// SIMATIC S7-200 project (STEP 7-Micro/WIN), CPU 226 CN REL 02.01

SYMBOL_TABLE 用户定义1
I_ERR1_QX        I4.2
I_ERR1_SF1       I0.0
I_ERR1_SF2       I0.1
I_ERR1_PF        I0.2
I_ERR1_JR        I0.3
I_TEST1_P        I0.4
I_L_ONOFF1       I0.5
I_ERR2_SF1       I0.7
I_ERR2_SF2       I1.0
I_ERR2_PF        I1.1
I_ERR2_JR        I1.2
I_TEST2_P        I1.3
I_L_ONOFF2       I1.4
I_ERR3_SF1       I1.6
I_ERR3_SF2       I1.7
I_ERR3_PF        I2.0
I_ERR3_JR        I2.1
I_TEST3_P        I2.2
I_L_ONOFF3       I2.3
I_ERR4_SF1       I2.5
I_ERR4_SF2       I2.6
I_ERR4_PF        I2.7
I_ERR4_JR        I3.0
I_TEST4_P        I3.1
I_L_ONOFF4       I3.2
I_MODE_CHANGE    I3.3
I_ONOFF1         I3.4
I_ONOFF2         I3.5
I_ONOFF3         I3.6
I_ONOFF4         I3.7
I_ONOFF          I4.0
I_JT             I4.1
I_ERR_WY         I4.5
I_ERR_GAS        I4.6
I_ERR_FIRE       I4.7
AQ_PF2           AQW0
AQ_PF4           AQW4
Q1_SF1           Q0.0
Q1_SF2           Q0.1
Q1_PF            Q0.2
Q1_JR            Q0.3
Q1_LIGHT         Q0.4
Q1_RUN           Q0.5
Q1_FM            Q0.6
Q1_PQ            Q0.7
Q1_KQ            Q1.0
Q2_SF1           Q1.1
Q2_SF2           Q1.2
Q2_PF            Q1.3
Q2_JR            Q1.4
Q2_LIGHT         Q1.5
Q2_RUN           Q1.6
Q2_FM            Q1.7
Q3_SF1           Q2.0
Q3_SF2           Q2.1
Q3_PF            Q2.2
Q3_JR            Q2.3
Q3_LIGHT         Q2.4
Q3_RUN           Q2.5
Q3_FM            Q2.6
Q4_SF1           Q3.0
Q4_SF2           Q3.1
Q4_PF            Q3.2
Q4_JR            Q3.3
Q4_LIGHT         Q3.4
Q4_RUN           Q3.5
Q4_FM            Q3.6
Q_RUN            Q3.7
F_HOUR_FLAG      M0.0
F_DELAY_WRITE    M0.1
F_DISSTART       M0.2
F_DISSTOP        M0.3
F_AUTO           M0.4
F_FILTER         M0.5
F_SAMPLING       M0.6
F_ERR            M0.7
F_NO_HMI         M1.0
F_S_ONOFF        M1.1
F_START          M1.2
F_STOP           M1.3
F_S_PQ           M1.4
F_S_GD           M1.5
F_S_KQ           M1.6
F_S_TOPPQ        M1.7
F_S_M_CHGE       M2.0
F_EN_M_CHGE      M2.1
F_TO_PQ          M2.2
F_TO_GD          M2.3
F_TO_KQ          M2.4
F_TO_TOPPQ       M2.5
F_GD_RESTART     M2.6
F_S_L_BOT_ONOFF  M2.7
F_RESTART_ALL    M3.0
F_ON_GAS         M3.1
F_RESET_START    M3.2
F_RESET_STOP     M3.3
F_RESET_OP_JR    M3.4
F_RESET_PAUSE    M3.5
F_RESET_RESTART  M3.6
F_RESET_RUN      M3.7
F_RESET_OPEN     M4.0
F_GD1            M4.1
F_GD2            M4.2
F_GD3            M4.3
F_GD4            M4.4
F_GD_END         M4.5
F_MODE_CHGE      M4.6
F_CHANGE         M4.7
F_DELAY_O_24     M5.0
F_Q_CHANGE       M5.1
F_S_ONOFF1       M7.0
F_START1         M7.1
F_STOP1          M7.2
F_S_L_ONOFF1     M7.3
F_ERR1           M7.4
F_RUN1           M7.5
F_OPEN1          M7.6
F_FLASH1         M7.7
F_FLASH1_ON      M8.0
F_PQ1_O_3S       M8.1
F_PQ1_O_6S       M8.2
F_PQ1_C_10S      M8.3
F_PQ1_C_5S       M8.4
F_KQ1_O_30S      M8.5
F_KQ1_O_3S       M8.6
F_KQ1_C_10S      M8.7
F_KQ1_C_5S       M9.0
F_PAUSE1         M9.1
F_RESTART1       M9.2
F1_OP_JR         M9.3
F_S_ONOFF2       M10.0
F_START2         M10.1
F_STOP2          M10.2
F_S_L_ONOFF2     M10.3
F_ERR2           M10.4
F_RUN2           M10.5
F_OPEN2          M10.6
F_FLASH2         M10.7
F_FLASH2_ON      M11.0
F_PQ2_O_3S       M11.1
F_PQ2_O_6S       M11.2
F_PQ2_C_10S      M11.3
F_PQ2_C_5S       M11.4
F_KQ2_O_30S      M11.5
F_KQ2_O_3S       M11.6
F_KQ2_C_10S      M11.7
F_KQ2_C_5S       M12.0
F_PAUSE2         M12.1
F_RESTART2       M12.2
F2_OP_JR         M12.3
F_S_ONOFF3       M13.0
F_START3         M13.1
F_STOP3          M13.2
F_S_L_ONOFF3     M13.3
F_ERR3           M13.4
F_RUN3           M13.5
F_OPEN3          M13.6
F_FLASH3         M13.7
F_FLASH3_ON      M14.0
F_PQ3_O_3S       M14.1
F_PQ3_O_6S       M14.2
F_PQ3_C_10S      M14.3
F_PQ3_C_5S       M14.4
F_KQ3_O_30S      M14.5
F_KQ3_O_3S       M14.6
F_KQ3_C_10S      M14.7
F_KQ3_C_5S       M15.0
F_PAUSE3         M15.1
F_RESTART3       M15.2
F3_OP_JR         M15.3
F_S_ONOFF4       M16.0
F_START4         M16.1
F_STOP4          M16.2
F_S_L_ONOFF4     M16.3
F_ERR4           M16.4
F_RUN4           M16.5
F_OPEN4          M16.6
F_FLASH4         M16.7
F_FLASH4_ON      M17.0
F_PQ4_O_3S       M17.1
F_PQ4_O_6S       M17.2
F_PQ4_C_10S      M17.3
F_PQ4_C_5S       M17.4
F_KQ4_O_30S      M17.5
F_KQ4_O_3S       M17.6
F_KQ4_C_10S      M17.7
F_KQ4_C_5S       M18.0
F_PAUSE4         M18.1
F_RESTART4       M18.2
F4_OP_JR         M18.3
F_S_ONOFF5       M19.0
F_START5         M19.1
F_STOP5          M19.2
F_S_L_ONOFF5     M19.3
F_ERR5           M19.4
F_RUN5           M19.5
F_OPEN5          M19.6
F_FLASH5         M19.7
F_FLASH5_ON      M20.0
F_PQ5_O_3S       M20.1
F_PQ5_O_6S       M20.2
F_PQ5_C_10S      M20.3
F_PQ5_C_5S       M20.4
F_KQ5_O_30S      M20.5
F_KQ5_O_3S       M20.6
F_KQ5_C_10S      M20.7
F_KQ5_C_5S       M21.0
F_PAUSE5         M21.1
F_RESTART5       M21.2
F5_OP_JR         M21.3
SYSTEM_ERROR_FLAG M23.2
Comu_Flag1       M23.3
Comu_Flag2       M23.4
Comu_Start       M23.5
Comu_End         M23.6
Real_Time        VW100
TEMP1_1          VW404
TEMP1_2          VW406
TEMP1_3          VW408
TEMP1_4          VW410
TEMP1_5          VW412
TEMP1_6          VW414
TEMP2_1          VW420
TEMP2_2          VW422
TEMP2_3          VW424
TEMP2_4          VW426
TEMP2_5          VW428
TEMP2_6          VW430
TEMP3_1          VW436
TEMP3_2          VW438
TEMP3_3          VW440
TEMP3_4          VW442
TEMP3_5          VW444
TEMP3_6          VW446
TEMP4_1          VW452
TEMP4_2          VW454
TEMP4_3          VW456
TEMP4_4          VW458
TEMP4_5          VW460
TEMP4_6          VW462
TEMP5_1          VW468
TEMP5_2          VW470
TEMP5_3          VW472
TEMP5_4          VW474
TEMP5_5          VW476
TEMP5_6          VW478
TEMP6_1          VW484
TEMP6_2          VW486
TEMP6_3          VW488
TEMP6_4          VW490
TEMP6_5          VW492
TEMP6_6          VW494
TEMP7_1          VW500
TEMP7_2          VW502
TEMP7_3          VW504
TEMP7_4          VW506
TEMP7_5          VW508
TEMP7_6          VW510
TEMP8_1          VW516
TEMP8_2          VW518
TEMP8_3          VW520
TEMP8_4          VW522
TEMP8_5          VW524
TEMP8_6          VW526
TEMP9_1          VW532
TEMP9_2          VW534
TEMP9_3          VW536
TEMP9_4          VW538
TEMP9_5          VW540
TEMP9_6          VW542
TEMP10_1         VW548
TEMP10_2         VW550
TEMP10_3         VW552
TEMP10_4         VW554
TEMP10_5         VW556
TEMP10_6         VW558
TEMP11_1         VW564
TEMP11_2         VW566
TEMP11_3         VW568
TEMP11_4         VW570
TEMP11_5         VW572
TEMP11_6         VW574
TEMP12_1         VW580
TEMP12_2         VW582
TEMP12_3         VW584
TEMP12_4         VW586
TEMP12_5         VW588
TEMP12_6         VW590
TEMP13_1         VW596
TEMP13_2         VW598
TEMP13_3         VW600
TEMP13_4         VW602
TEMP13_5         VW604
TEMP13_6         VW606
TEMP14_1         VW612
TEMP14_2         VW614
TEMP14_3         VW616
TEMP14_4         VW618
TEMP14_5         VW620
TEMP14_6         VW622
TEMP15_1         VW628
TEMP15_2         VW630
TEMP15_3         VW632
TEMP15_4         VW634
TEMP15_5         VW636
TEMP15_6         VW638
TEMP16_1         VW644
TEMP16_2         VW646
TEMP16_3         VW648
TEMP16_4         VW650
TEMP16_5         VW652
TEMP16_6         VW654
T_ERRL           VW700
T_ERRH           VW702
T_SAMPLING       VW704
ADDR_EEP         VW706
TEMP_PQ_H        VW708
TEMP_PQ_L        VW710
TEMP_PQ_ALARM_T1 VW712
TEMP_PQ_ALARM_T2 VW714
TEMP_KQ_H        VW716
TEMP_KQ_L        VW718
TEMP_KQ_ALARM_T1 VW720
TEMP_KQ_ALARM_T2 VW722
TIME_PQ          VW724
TIME_KQ          VW726
TIME_LQ          VW728
DELAY_START      VW730
TIME_DOOR        VW732
TEMP_H           VW754
TEMP_L           VW756
TEMP_T1_ALARM    VW758
TEMP_T2_ALARM    VW760
DELAY_C_PQ       VW762
DELAY_C_KQ       VW764
T_RUN            VW766
DELAY_O_24       VW768
DELAY_FM         VW770
C_ONOFF          VB800
C_ERR_HMI        VB801
C_SAMPLING       VB802
AD_ADDR          VB803
C_KEY            VB804
C_ERR            VB805
C_ERR_FIRE       VB806
C_ERR_WY         VB807
C_ERR_GAS        VB808
C_JT             VB809
C_PQ             VB810
C_GD             VB811
C_KQ             VB812
C_TOPPQ          VB813
C_M_CHGE         VB814
C_L_BOT_ONOFF    VB815
C_GD1            VB816
C_GD2            VB817
C_GD3            VB818
C_GD4            VB819
C_GD_END         VB820
C_ONOFF1         VB821
C_ERR1_QX        VB822
C_ERR1_SF1       VB823
C_ERR1_SF2       VB824
C_ERR1_PF        VB825
C_ERR1_JR        VB826
C_ERR1_T1        VB827
C_ERR1_T2        VB828
C_OVER1_T1       VB829
C_OVER1_T2       VB830
C_TEST1_P        VB831
C_L_ONOFF1       VB832
EX_MODE          VB833
REAL_MODE        VB834
TEMP_MODE        VB835
C_ONOFF2         VB840
C_L_ONOFF2       VB841
C_ERR2_QX        VB842
C_ERR2_SF1       VB843
C_ERR2_SF2       VB844
C_ERR2_PF        VB845
C_ERR2_JR        VB846
C_ERR2_T1        VB847
C_ERR2_T2        VB848
C_OVER2_T1       VB849
C_OVER2_T2       VB850
C_TEST2_P        VB851
C_ONOFF3         VB860
C_L_ONOFF3       VB861
C_ERR3_QX        VB862
C_ERR3_SF1       VB863
C_ERR3_SF2       VB864
C_ERR3_PF        VB865
C_ERR3_JR        VB866
C_ERR3_T1        VB867
C_ERR3_T2        VB868
C_OVER3_T1       VB869
C_OVER3_T2       VB870
C_TEST3_P        VB871
C_ONOFF4         VB880
C_L_ONOFF4       VB881
C_ERR4_QX        VB882
C_ERR4_SF1       VB883
C_ERR4_SF2       VB884
C_ERR4_PF        VB885
C_ERR4_JR        VB886
C_ERR4_T1        VB887
C_ERR4_T2        VB888
C_OVER4_T1       VB889
C_OVER4_T2       VB890
C_TEST4_P        VB891
C_ONOFF5         VB900
C_L_ONOFF5       VB901
C_ERR5_QX        VB902
C_ERR5_SF1       VB903
C_ERR5_SF2       VB904
C_ERR5_PF        VB905
C_ERR5_JR        VB906
C_ERR5_T1        VB907
C_ERR5_T2        VB908
C_OVER5_T1       VB909
C_OVER5_T2       VB910
C_TEST5_P        VB911
MEASURE_MODE     VB914
C_ERR_W1         VW822
C_ERR_W2         VW842
C_ERR_W3         VW862
C_ERR_W4         VW882
C_ERR_W5         VW902
ERR1_1           VB1000
F_ERR1_QX        V1000.0
F_ERR1_SF1       V1000.1
F_ERR1_SF2       V1000.2
F_ERR1_PF        V1000.3
F_ERR1_JR        V1000.4
F_ERR1_P         V1000.5
ERR1_2           VB1001
F_ERR1_T1        V1001.0
F_ERR1_T2        V1001.1
F_OVER1_T1       V1001.2
F_OVER1_T2       V1001.3
ERR2_1           VB1002
F_ERR2_QX        V1002.0
F_ERR2_SF1       V1002.1
F_ERR2_SF2       V1002.2
F_ERR2_PF        V1002.3
F_ERR2_JR        V1002.4
F_ERR2_P         V1002.5
ERR2_2           VB1003
F_ERR2_T1        V1003.0
F_ERR2_T2        V1003.1
F_OVER2_T1       V1003.2
F_OVER2_T2       V1003.3
ERR3_1           VB1004
F_ERR3_QX        V1004.0
F_ERR3_SF1       V1004.1
F_ERR3_SF2       V1004.2
F_ERR3_PF        V1004.3
F_ERR3_JR        V1004.4
F_ERR3_P         V1004.5
ERR3_2           VB1005
F_ERR3_T1        V1005.0
F_ERR3_T2        V1005.1
F_OVER3_T1       V1005.2
F_OVER3_T2       V1005.3
ERR4_1           VB1006
F_ERR4_QX        V1006.0
F_ERR4_SF1       V1006.1
F_ERR4_SF2       V1006.2
F_ERR4_PF        V1006.3
F_ERR4_JR        V1006.4
F_ERR4_P         V1006.5
ERR4_2           VB1007
F_ERR4_T1        V1007.0
F_ERR4_T2        V1007.1
F_OVER4_T1       V1007.2
F_OVER4_T2       V1007.3
ERR5_1           VB1008
F_ERR5_QX        V1008.0
F_ERR5_SF1       V1008.1
F_ERR5_SF2       V1008.2
F_ERR5_PF        V1008.3
F_ERR5_JR        V1008.4
F_ERR5_P         V1008.5
ERR5_2           VB1009
F_ERR5_T1        V1009.0
F_ERR5_T2        V1009.1
F_OVER5_T1       V1009.2
F_OVER5_T2       V1009.3
EN_QX            VB1010
F_EN_QX1         V1010.0
F_EN_QX2         V1010.1
F_EN_QX3         V1010.2
F_EN_QX4         V1010.3
F_EN_QX5         V1010.4
EN_OP1           VB1011
F_EN_ON_ALL      V1011.0
F_EN_OFF_ALL     V1011.1
F_EN_ON_1        V1011.2
F_EN_OFF_1       V1011.3
F_EN_ON_2        V1011.4
F_EN_OFF_2       V1011.5
F_EN_ON_3        V1011.6
F_EN_OFF_3       V1011.7
EN_OP2           VB1012
F_EN_ON_4        V1012.0
F_EN_OFF_4       V1012.1
F_EN_ON_5        V1012.2
F_EN_OFF_5       V1012.3
STATE            VB1014
F_STATE1         V1014.0
F_STATE2         V1014.1
F_STATE3         V1014.2
F_STATE4         V1014.3
F_STATE5         V1014.4
MINUTE           VB1016
ERR_MOUDLE       VB1017
F_ERR_MK1        V1017.0
F_ERR_MK2        V1017.1
F_ERR_MK3        V1017.2
F_ERR_MK4        V1017.3
F_ERR_MK5        V1017.4
F_ERR_MK6        V1017.5
DELAY            VB1018
INPUT_JT         VB1019
F_JT             V1019.0
OIL_ERROR        V1019.1
OIL_ERROR_H      V1019.2
EN_CHANGE        VB1020
F_EN_CHGE1       V1020.0
F_EN_CHGE2       V1020.1
F_EN_CHGE3       V1020.2
F_EN_CHGE4       V1020.3
F_EN_CHGE5       V1020.4
ERR              VB1021
F_ERR_GAS        V1021.0
F_ERR_WY         V1021.1
F_ERR_FIRE       V1021.2
DO_SF1_PC1       V1022.0
DO_SF2_PC1       V1022.1
DO_PF_PC1        V1022.2
DO_HEAT_PC1      V1022.3
DO_FM_PC1        V1022.4
DO_SF1_PC2       V1022.5
DO_SF2_PC2       V1022.6
DO_PF_PC2        V1022.7
DO_HEAT_PC2      V1023.0
DO_FM_PC2        V1023.1
DO_SF1_PC3       V1023.2
DO_SF2_PC3       V1023.3
DO_PF_PC3        V1023.4
DO_HEAT_PC3      V1023.5
DO_FM_PC3        V1023.6
DO_SF1_PC4       V1023.7
DO_SF2_PC4       V1024.0
DO_PF_PC4        V1024.1
DO_HEAT_PC4      V1024.2
DO_FM_PC4        V1024.3
DO_SF1_PC5       V1024.4
DO_SF2_PC5       V1024.5
DO_PF_PC5        V1024.6
DO_HEAT_PC5      V1024.7
DO_FM_PC5        V1025.0
TE1_SENSOR1      VW1050
TE1_SENSOR2      VW1052
TE2_SENSOR1      VW1054
TE2_SENSOR2      VW1056
TE3_SENSOR1      VW1058
TE3_SENSOR2      VW1060
TE4_SENSOR1      VW1062
TE4_SENSOR2      VW1064
TE5_SENSOR1      VW1066
TE5_SENSOR2      VW1068
RUN1             VW1070
RUN2             VW1072
RUN3             VW1074
RUN4             VW1076
RUN5             VW1078
I_A              VW1080
I_B              VW1082
I_C              VW1084
I2_PF            VW1086
I4_PF            VW1088
OIL_REAL         VW1090
OIL_VALUE_SCREEN VW1092
SET_PQ           VB1100
SET_WX_PQ        VB1101
OIL_ENABLE       VB1102
SET_KQ           VB1103
SET_WX_KQ        VB1104
SET_T2_ALARM     VB1105
SET_DELAY_PQ     VB1106
SET_DELAY_KQ     VB1107
SET_DELAY_O24    VB1108
FM_DELAY_TIME    VB1109
SET_PQ_RUNTIME   VW1110
SET_KQ_RUNTIME   VW1112
SET_I2_PF_PQ     VB1114
SET_I4_PF_PQ     VB1115
SET_I2_PF_GD     VB1116
SET_I4_PF_GD     VB1117
OIL_SET          VW1118
SET_DELAY_KQ2    VW1120
SET1_TEMP1_20    VW1122
SET2_TEMP1_20    VW1124
SET3_TEMP1_20    VW1126
SET4_TEMP1_20    VW1128
SET5_TEMP1_20    VW1130
SET1_TEMP2_20    VW1132
SET2_TEMP2_20    VW1134
SET3_TEMP2_20    VW1136
SET4_TEMP2_20    VW1138
SET5_TEMP2_20    VW1140
OIL_SET_H        VW1146
CTRL_WORKSTATE   VB1150
HMI_COMM         VB1151
CTRL_CLRQX       VB1152
F1_CLRQX         V1152.0
F2_CLRQX         V1152.1
F3_CLRQX         V1152.2
F4_CLRQX         V1152.3
F5_CLRQX         V1152.4
CTRL_ONOFF1      VB1153
F_CTRL_ALL_ON    V1153.0
F_CTRL_ALL_OFF   V1153.1
F_CTRL1_ON       V1153.2
F_CTRL1_OFF      V1153.3
F_CTRL2_ON       V1153.4
F_CTRL2_OFF      V1153.5
F_CTRL3_ON       V1153.6
F_CTRL3_OFF      V1153.7
CTRL_ONOFF2      VB1154
F_CTRL4_ON       V1154.0
F_CTRL4_OFF      V1154.1
F_CTRL5_ON       V1154.2
F_CTRL5_OFF      V1154.3
CTRL_MODE        VB1155
SET_TEM1         VB1156
F_SET1_TEM1      V1156.0
F_SET2_TEM1      V1156.1
F_SET3_TEM1      V1156.2
F_SET4_TEM1      V1156.3
F_SET5_TEM1      V1156.4
SET_TEM2         VB1157
F_SET1_TEM2      V1157.0
F_SET2_TEM2      V1157.1
F_SET3_TEM2      V1157.2
F_SET4_TEM2      V1157.3
F_SET5_TEM2      V1157.4
SAVE_PQ          VB1700
SAVE_WX_PQ       VB1701
SAVE_KQ          VB1703
SAVE_WX_KQ       VB1704
SAVE_T2_ALARM    VB1705
SAVE_DELAY_PQ    VB1706
SAVE_DELAY_KQ    VB1707
SAVE_DELAY_O24   VB1708
SAVE_DELAY_FM    VB1709
SAVE_PQ_RUNTIME  VW1710
SAVE_KQ_RUNTIME  VW1712
SAVE_I2_PF_PQ    VB1714
SAVE_I4_PF_PQ    VB1715
SAVE_I2_PF_GD    VB1716
SAVE_I4_PF_GD    VB1717
SAVE_I2_PF_KQ    VB1718
SAVE_I4_PF_KQ    VB1719
SAVE_DELAY_KQ2   VW1720
SAVE1_TEMP1_20   VW1722
SAVE2_TEMP1_20   VW1724
SAVE3_TEMP1_20   VW1726
SAVE4_TEMP1_20   VW1728
SAVE5_TEMP1_20   VW1730
SAVE1_TEMP2_20   VW1732
SAVE2_TEMP2_20   VW1734
SAVE3_TEMP2_20   VW1736
SAVE4_TEMP2_20   VW1738
SAVE5_TEMP2_20   VW1740
RUN_TIME_CAL     VD920
RUN_TIME_ALL     VD1142
END_SYMBOL_TABLE

SYMBOL_TABLE S7-200 符号
Always_On        SM0.0    // 始终接通为 ON
First_Scan_On    SM0.1    // 仅第一个扫描周期中接通为 ON
Clock_1s         SM0.5    // 在 1 秒钟的循环周期内，接通为 ON 0.5 秒，关断为 OFF 0.5  秒
P0_Ctrl_Rcv_7    SM87.7   // 0 = 信息接收功能被禁止，1 = 信息接收功能被使能
EM0_ID           SMB8     // 模块 0 识别（ID）寄存器
EM0_Err          SMB9     // 模块 0 错误寄存器
EM1_ID           SMB10    // 模块 1 识别（ID）寄存器
EM1_Err          SMB11    // 模块 1 错误寄存器
EM2_ID           SMB12    // 模块 2 识别（ID）寄存器
EM2_Err          SMB13    // 模块 2 错误寄存器
EM3_ID           SMB14    // 模块 3 识别（ID）寄存器
EM3_Err          SMB15    // 模块 3 错误寄存器
EM4_ID           SMB16    // 模块 4 识别（ID）寄存器
EM4_Err          SMB17    // 模块 4 错误寄存器
EM5_ID           SMB18    // 模块 5 识别（ID）寄存器
EM5_Err          SMB19    // 模块 5 错误寄存器
P0_Config        SMB30    // 通信端口 0 设置：奇偶校验、每个字符的数据位数目、波特率和协议
Save_to_EEPROM   SMB31    // 设置保存参数，以便将 V 存储区中的一个数据保存至永久性存储区（EEPROM）
P0_Ctrl_Rcv      SMB87    // 信息接收控制
P0_Start_Char    SMB88    // 信息起始字符
P0_Max_Char      SMB94    // 信息接收最大字符数（1 至 255 个字节）
P0_Timeout       SMW92    // 字符间/信息间定时器超时数值，以毫秒为单位表示
END_SYMBOL_TABLE

ORGANIZATION_BLOCK 主程序:OB1
TITLE=程序注释
VAR
TEMP_B:BYTE;	// LB0 
TEMP_W:WORD;	// LW1 
TEMP_FLAG:BOOL;	// L3.0 
TEMP_B4:BYTE;	// LB4 
TEMP_B2:BYTE;	// LB5 
TEMP_W2:WORD;	// LW6 
END_VAR
BEGIN
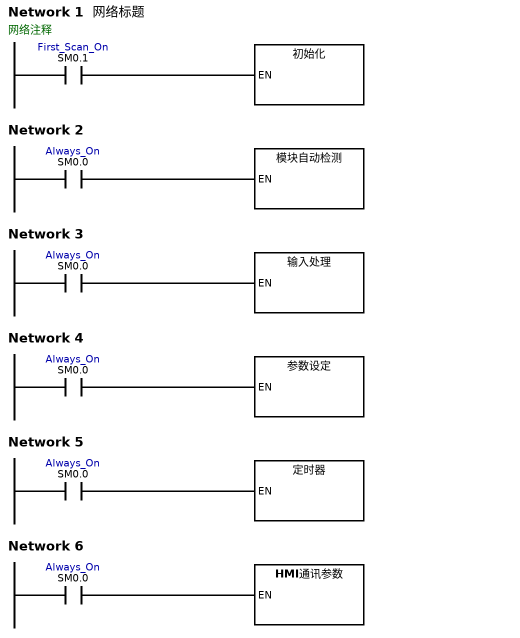
Network 1 // 网络标题
// 网络注释
LD     First_Scan_On:SM0.1
CALL   初始化:SBR1
Network 2
LD     Always_On:SM0.0
CALL   模块自动检测:SBR2
Network 3
LD     Always_On:SM0.0
CALL   输入处理:SBR3
Network 4
LD     Always_On:SM0.0
CALL   参数设定:SBR5
Network 5
LD     Always_On:SM0.0
CALL   定时器:SBR9
Network 6
LD     Always_On:SM0.0
CALL   HMI通讯参数:SBR4
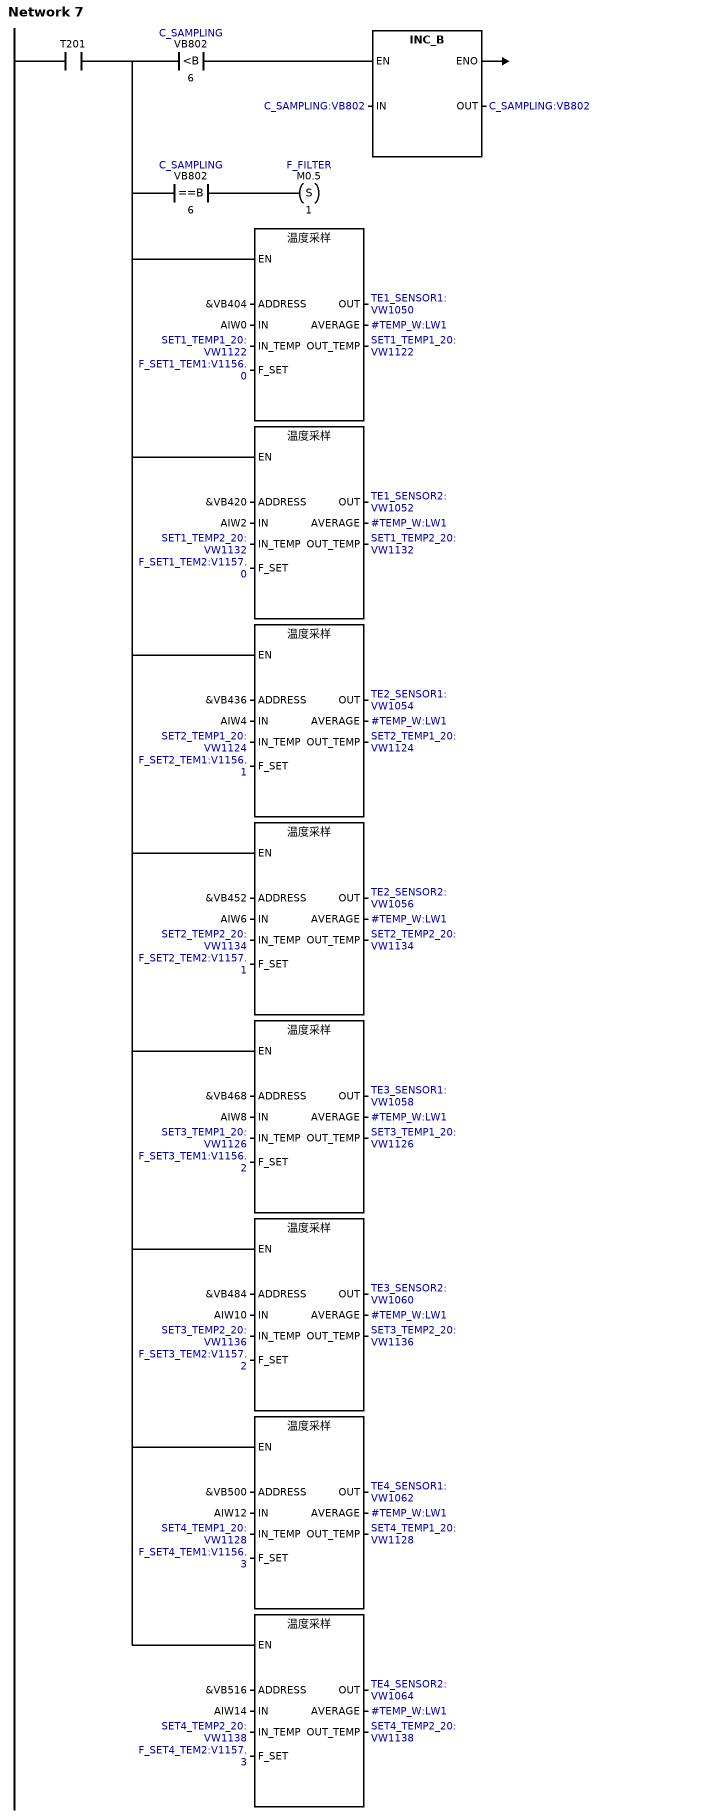
Network 7
LD     T201
LPS
AB<    C_SAMPLING:VB802, 6
INCB   C_SAMPLING:VB802
LRD
AB=    C_SAMPLING:VB802, 6
S      F_FILTER:M0.5, 1
LRD
CALL   温度采样:SBR6, &VB404, AIW0, SET1_TEMP1_20:VW1122, F_SET1_TEM1:V1156.0, TE1_SENSOR1:VW1050, #TEMP_W:LW1, SET1_TEMP1_20:VW1122
LRD
CALL   温度采样:SBR6, &VB420, AIW2, SET1_TEMP2_20:VW1132, F_SET1_TEM2:V1157.0, TE1_SENSOR2:VW1052, #TEMP_W:LW1, SET1_TEMP2_20:VW1132
LRD
CALL   温度采样:SBR6, &VB436, AIW4, SET2_TEMP1_20:VW1124, F_SET2_TEM1:V1156.1, TE2_SENSOR1:VW1054, #TEMP_W:LW1, SET2_TEMP1_20:VW1124
LRD
CALL   温度采样:SBR6, &VB452, AIW6, SET2_TEMP2_20:VW1134, F_SET2_TEM2:V1157.1, TE2_SENSOR2:VW1056, #TEMP_W:LW1, SET2_TEMP2_20:VW1134
LRD
CALL   温度采样:SBR6, &VB468, AIW8, SET3_TEMP1_20:VW1126, F_SET3_TEM1:V1156.2, TE3_SENSOR1:VW1058, #TEMP_W:LW1, SET3_TEMP1_20:VW1126
LRD
CALL   温度采样:SBR6, &VB484, AIW10, SET3_TEMP2_20:VW1136, F_SET3_TEM2:V1157.2, TE3_SENSOR2:VW1060, #TEMP_W:LW1, SET3_TEMP2_20:VW1136
LRD
CALL   温度采样:SBR6, &VB500, AIW12, SET4_TEMP1_20:VW1128, F_SET4_TEM1:V1156.3, TE4_SENSOR1:VW1062, #TEMP_W:LW1, SET4_TEMP1_20:VW1128
LPP
CALL   温度采样:SBR6, &VB516, AIW14, SET4_TEMP2_20:VW1138, F_SET4_TEM2:V1157.3, TE4_SENSOR2:VW1064, #TEMP_W:LW1, SET4_TEMP2_20:VW1138
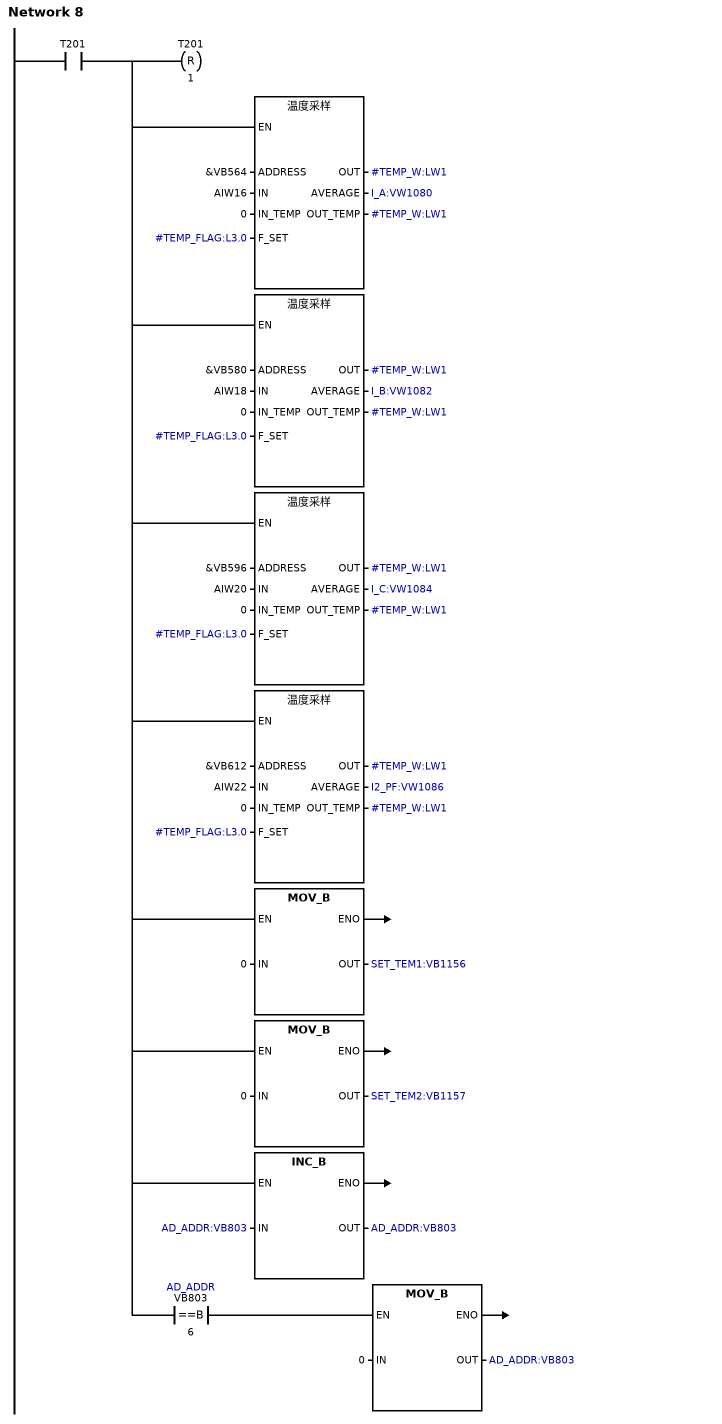
Network 8
LD     T201
R      T201, 1
CALL   温度采样:SBR6, &VB564, AIW16, 0, #TEMP_FLAG:L3.0, #TEMP_W:LW1, I_A:VW1080, #TEMP_W:LW1
CALL   温度采样:SBR6, &VB580, AIW18, 0, #TEMP_FLAG:L3.0, #TEMP_W:LW1, I_B:VW1082, #TEMP_W:LW1
CALL   温度采样:SBR6, &VB596, AIW20, 0, #TEMP_FLAG:L3.0, #TEMP_W:LW1, I_C:VW1084, #TEMP_W:LW1
CALL   温度采样:SBR6, &VB612, AIW22, 0, #TEMP_FLAG:L3.0, #TEMP_W:LW1, I2_PF:VW1086, #TEMP_W:LW1
MOVB   0, SET_TEM1:VB1156
MOVB   0, SET_TEM2:VB1157
INCB   AD_ADDR:VB803
AB=    AD_ADDR:VB803, 6
MOVB   0, AD_ADDR:VB803
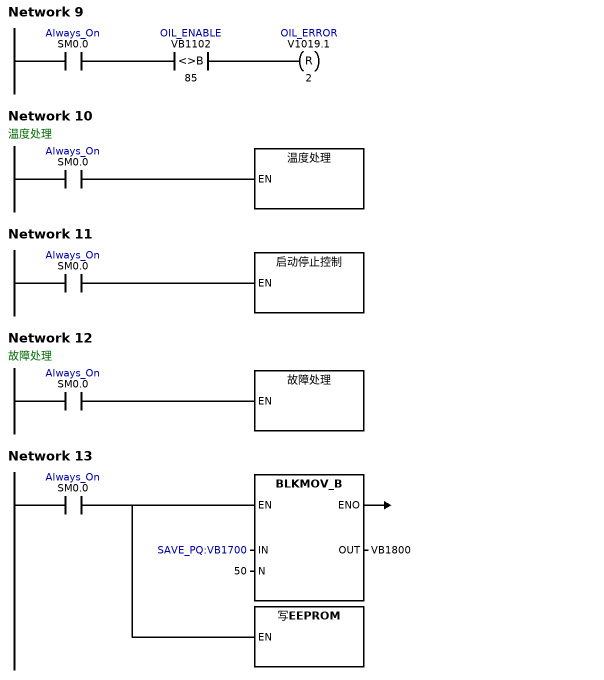
Network 9
LD     Always_On:SM0.0
AB<>   OIL_ENABLE:VB1102, 85
R      OIL_ERROR:V1019.1, 2
Network 10
// 温度处理
LD     Always_On:SM0.0
CALL   温度处理:SBR10
Network 11
LD     Always_On:SM0.0
CALL   启动停止控制:SBR7
Network 12
// 故障处理
LD     Always_On:SM0.0
CALL   故障处理:SBR11
Network 13
LD     Always_On:SM0.0
BMB    SAVE_PQ:VB1700, VB1800, 50
CALL   写EEPROM:SBR19
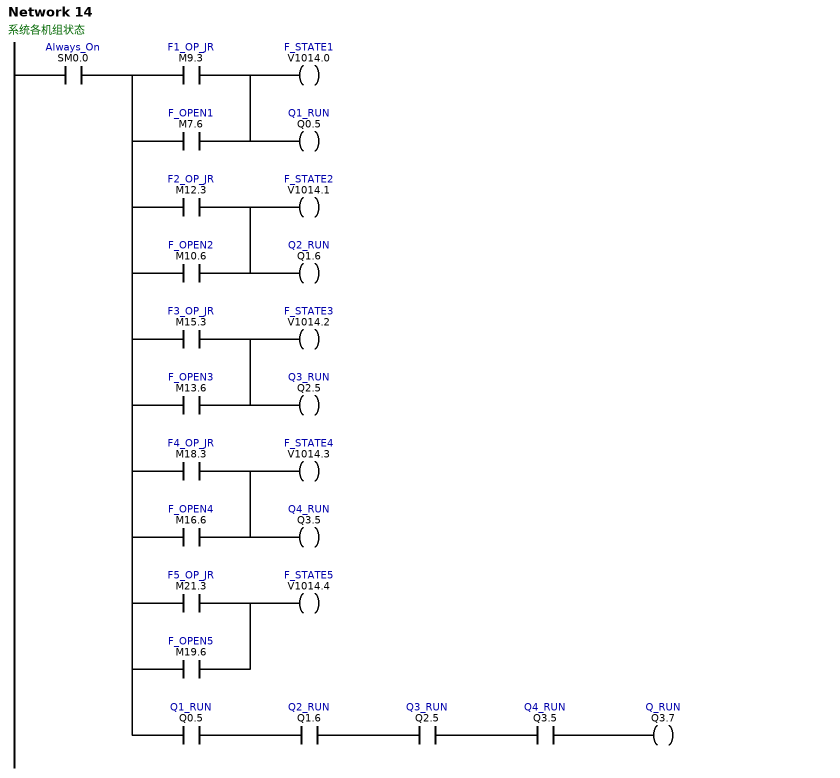
Network 14
// 系统各机组状态
LD     Always_On:SM0.0
LPS
LD     F1_OP_JR:M9.3
O      F_OPEN1:M7.6
ALD
=      F_STATE1:V1014.0
=      Q1_RUN:Q0.5
LRD
LD     F2_OP_JR:M12.3
O      F_OPEN2:M10.6
ALD
=      F_STATE2:V1014.1
=      Q2_RUN:Q1.6
LRD
LD     F3_OP_JR:M15.3
O      F_OPEN3:M13.6
ALD
=      F_STATE3:V1014.2
=      Q3_RUN:Q2.5
LRD
LD     F4_OP_JR:M18.3
O      F_OPEN4:M16.6
ALD
=      F_STATE4:V1014.3
=      Q4_RUN:Q3.5
LRD
LD     F5_OP_JR:M21.3
O      F_OPEN5:M19.6
ALD
=      F_STATE5:V1014.4
LPP
A      Q1_RUN:Q0.5
A      Q2_RUN:Q1.6
A      Q3_RUN:Q2.5
A      Q4_RUN:Q3.5
=      Q_RUN:Q3.7
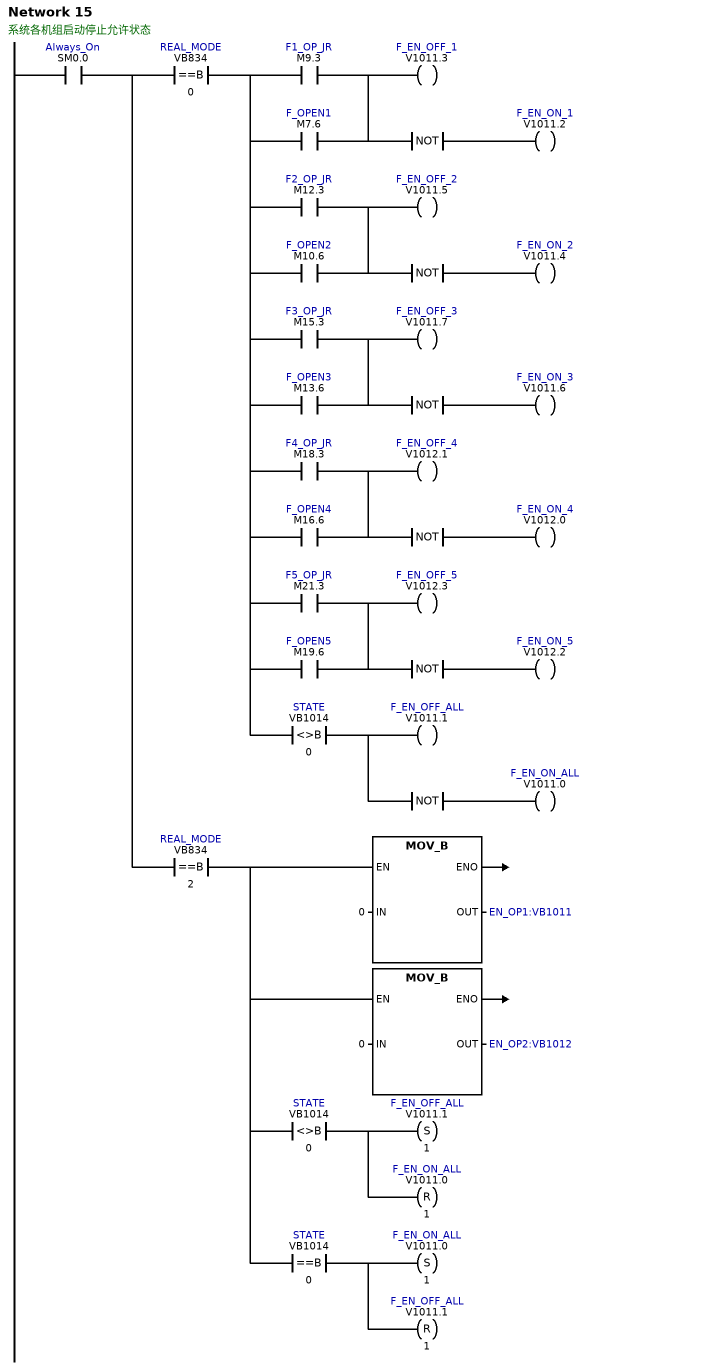
Network 15
// 系统各机组启动停止允许状态
LD     Always_On:SM0.0
LPS
AB=    REAL_MODE:VB834, 0
LPS
LD     F1_OP_JR:M9.3
O      F_OPEN1:M7.6
ALD
=      F_EN_OFF_1:V1011.3
NOT
=      F_EN_ON_1:V1011.2
LRD
LD     F2_OP_JR:M12.3
O      F_OPEN2:M10.6
ALD
=      F_EN_OFF_2:V1011.5
NOT
=      F_EN_ON_2:V1011.4
LRD
LD     F3_OP_JR:M15.3
O      F_OPEN3:M13.6
ALD
=      F_EN_OFF_3:V1011.7
NOT
=      F_EN_ON_3:V1011.6
LRD
LD     F4_OP_JR:M18.3
O      F_OPEN4:M16.6
ALD
=      F_EN_OFF_4:V1012.1
NOT
=      F_EN_ON_4:V1012.0
LRD
LD     F5_OP_JR:M21.3
O      F_OPEN5:M19.6
ALD
=      F_EN_OFF_5:V1012.3
NOT
=      F_EN_ON_5:V1012.2
LPP
AB<>   STATE:VB1014, 0
=      F_EN_OFF_ALL:V1011.1
NOT
=      F_EN_ON_ALL:V1011.0
LPP
AB=    REAL_MODE:VB834, 2
LPS
MOVB   0, EN_OP1:VB1011
MOVB   0, EN_OP2:VB1012
AB<>   STATE:VB1014, 0
S      F_EN_OFF_ALL:V1011.1, 1
R      F_EN_ON_ALL:V1011.0, 1
LPP
AB=    STATE:VB1014, 0
S      F_EN_ON_ALL:V1011.0, 1
R      F_EN_OFF_ALL:V1011.1, 1
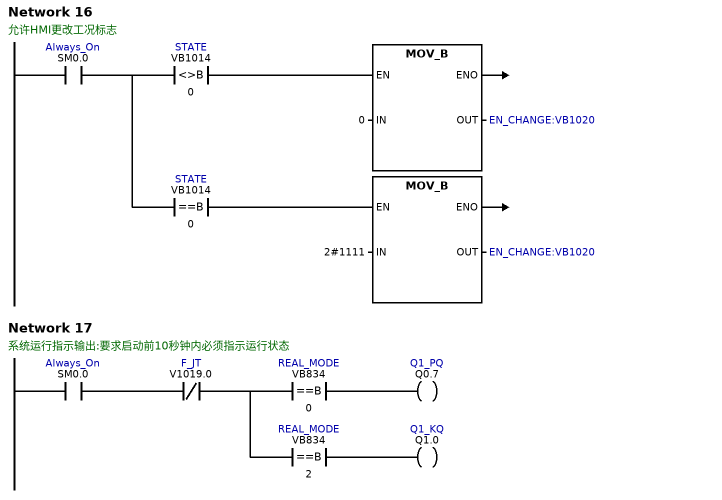
Network 16
// 允许HMI更改工况标志
LD     Always_On:SM0.0
LPS
AB<>   STATE:VB1014, 0
MOVB   0, EN_CHANGE:VB1020
LPP
AB=    STATE:VB1014, 0
MOVB   2#1111, EN_CHANGE:VB1020
Network 17
// 系统运行指示输出:要求启动前10秒钟内必须指示运行状态
LD     Always_On:SM0.0
AN     F_JT:V1019.0
LPS
AB=    REAL_MODE:VB834, 0
=      Q1_PQ:Q0.7
LPP
AB=    REAL_MODE:VB834, 2
=      Q1_KQ:Q1.0
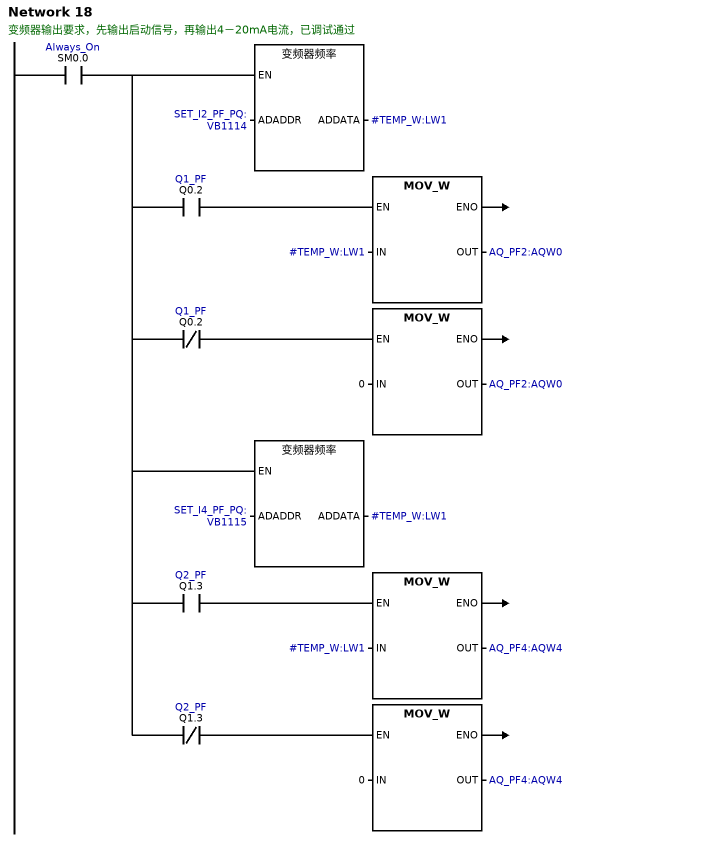
Network 18
// 变频器输出要求，先输出启动信号，再输出4－20mA电流，已调试通过
LD     Always_On:SM0.0
LPS
CALL   变频器频率:SBR12, SET_I2_PF_PQ:VB1114, #TEMP_W:LW1
A      Q1_PF:Q0.2
MOVW   #TEMP_W:LW1, AQ_PF2:AQW0
LRD
AN     Q1_PF:Q0.2
MOVW   0, AQ_PF2:AQW0
LRD
CALL   变频器频率:SBR12, SET_I4_PF_PQ:VB1115, #TEMP_W:LW1
LRD
A      Q2_PF:Q1.3
MOVW   #TEMP_W:LW1, AQ_PF4:AQW4
LPP
AN     Q2_PF:Q1.3
MOVW   0, AQ_PF4:AQW4
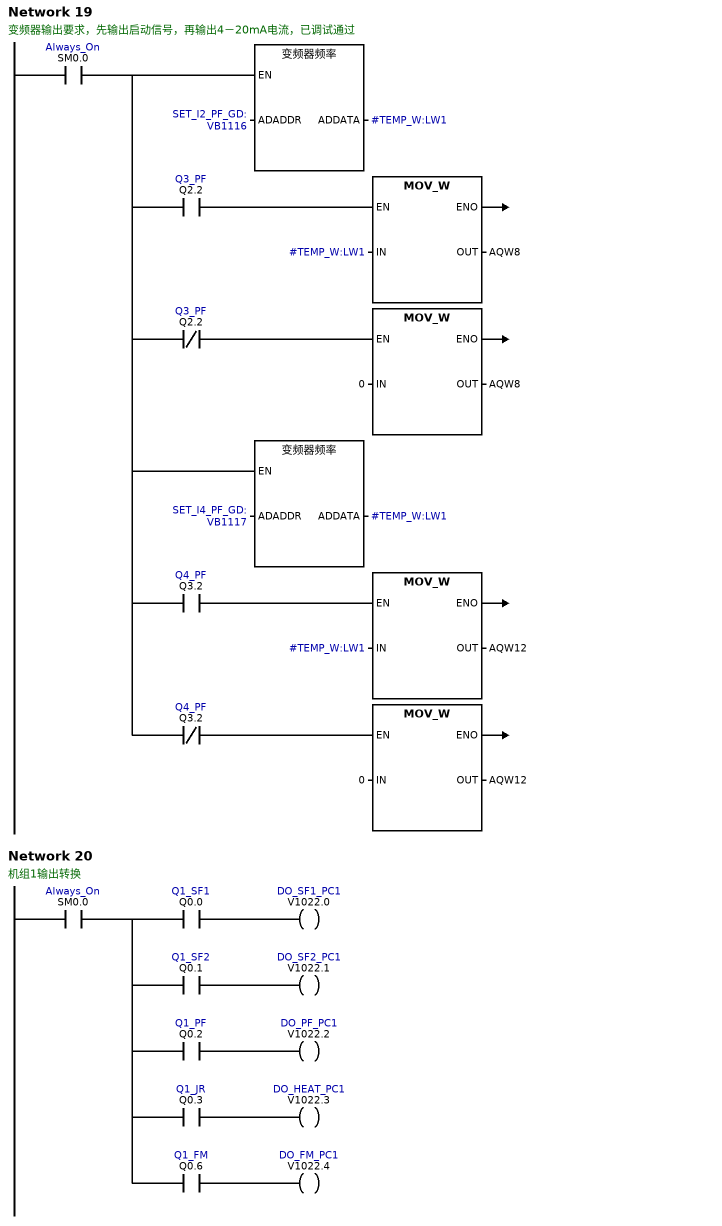
Network 19
// 变频器输出要求，先输出启动信号，再输出4－20mA电流，已调试通过
LD     Always_On:SM0.0
LPS
CALL   变频器频率:SBR12, SET_I2_PF_GD:VB1116, #TEMP_W:LW1
A      Q3_PF:Q2.2
MOVW   #TEMP_W:LW1, AQW8
LRD
AN     Q3_PF:Q2.2
MOVW   0, AQW8
LRD
CALL   变频器频率:SBR12, SET_I4_PF_GD:VB1117, #TEMP_W:LW1
LRD
A      Q4_PF:Q3.2
MOVW   #TEMP_W:LW1, AQW12
LPP
AN     Q4_PF:Q3.2
MOVW   0, AQW12
Network 20
// 机组1输出转换
LD     Always_On:SM0.0
LPS
A      Q1_SF1:Q0.0
=      DO_SF1_PC1:V1022.0
LRD
A      Q1_SF2:Q0.1
=      DO_SF2_PC1:V1022.1
LRD
A      Q1_PF:Q0.2
=      DO_PF_PC1:V1022.2
LRD
A      Q1_JR:Q0.3
=      DO_HEAT_PC1:V1022.3
LPP
A      Q1_FM:Q0.6
=      DO_FM_PC1:V1022.4
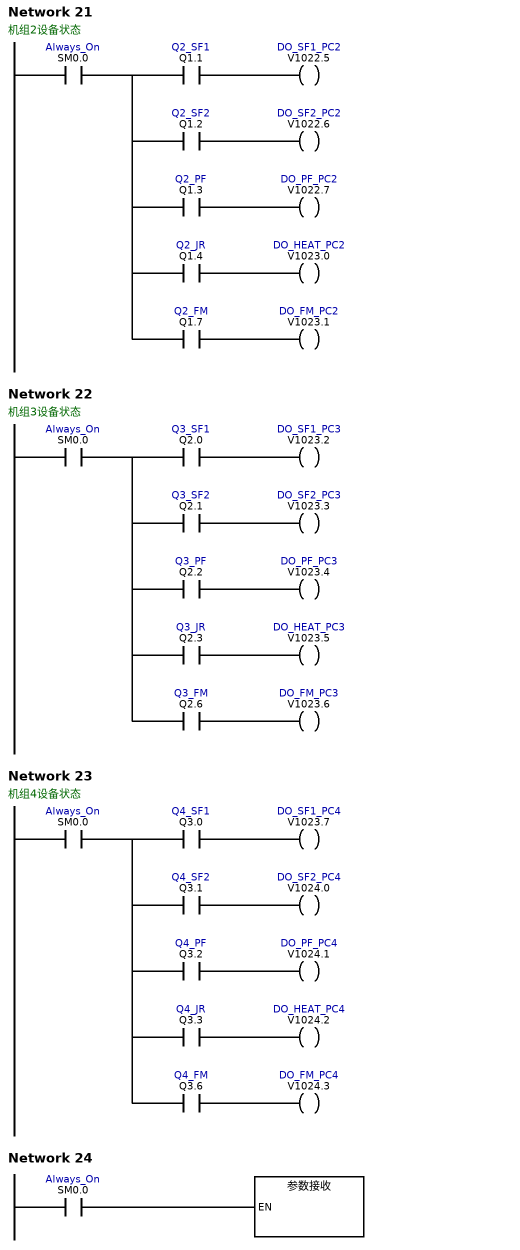
Network 21
// 机组2设备状态
LD     Always_On:SM0.0
LPS
A      Q2_SF1:Q1.1
=      DO_SF1_PC2:V1022.5
LRD
A      Q2_SF2:Q1.2
=      DO_SF2_PC2:V1022.6
LRD
A      Q2_PF:Q1.3
=      DO_PF_PC2:V1022.7
LRD
A      Q2_JR:Q1.4
=      DO_HEAT_PC2:V1023.0
LPP
A      Q2_FM:Q1.7
=      DO_FM_PC2:V1023.1
Network 22
// 机组3设备状态
LD     Always_On:SM0.0
LPS
A      Q3_SF1:Q2.0
=      DO_SF1_PC3:V1023.2
LRD
A      Q3_SF2:Q2.1
=      DO_SF2_PC3:V1023.3
LRD
A      Q3_PF:Q2.2
=      DO_PF_PC3:V1023.4
LRD
A      Q3_JR:Q2.3
=      DO_HEAT_PC3:V1023.5
LPP
A      Q3_FM:Q2.6
=      DO_FM_PC3:V1023.6
Network 23
// 机组4设备状态
LD     Always_On:SM0.0
LPS
A      Q4_SF1:Q3.0
=      DO_SF1_PC4:V1023.7
LRD
A      Q4_SF2:Q3.1
=      DO_SF2_PC4:V1024.0
LRD
A      Q4_PF:Q3.2
=      DO_PF_PC4:V1024.1
LRD
A      Q4_JR:Q3.3
=      DO_HEAT_PC4:V1024.2
LPP
A      Q4_FM:Q3.6
=      DO_FM_PC4:V1024.3
Network 24
LD     Always_On:SM0.0
CALL   参数接收:SBR0
END_ORGANIZATION_BLOCK

SUBROUTINE_BLOCK 参数接收:SBR0
TITLE=子程序注释
BEGIN
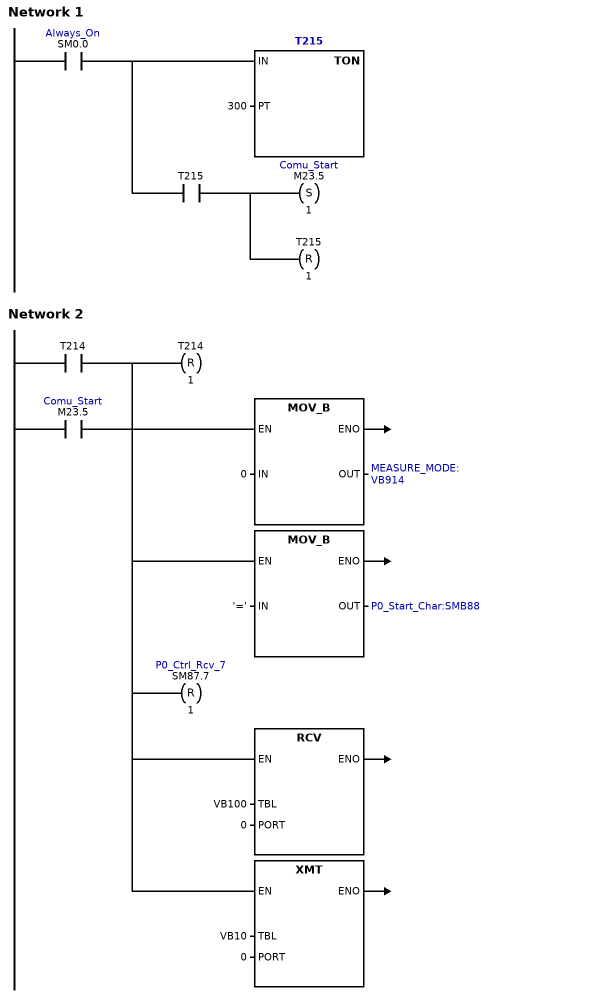
Network 1
// (network saved uncompiled; LAD cells follow)
// row 0: c0 -| |- Always_On:SM0.0 v  c1 --  c2 [TON T215 IN:=power@row0, PT:=300]
// row 1: c0 ^v  c2 [box]
// row 2: c0 ^  c1 -| |- T215 v  c2 -(S) Comu_Start:M23.5, 1
// row 3: c1 ^  c2 -(R) T215, 1
Network 2
// (network saved uncompiled; LAD cells follow)
// row 0: c0 -| |- T214 v  c1 -(R) T214, 1
// row 1: c0 -| |- Comu_Start:M23.5 ^v  c1 --  c2 [MOV_B EN:=power@row1, IN:=0, ENO=>power, OUT=>MEASURE_MODE:VB914]  c3 ->
// row 2: c0 ^v  c2 [box]
// row 3: c0 ^v  c1 --  c2 [MOV_B EN:=power@row3, IN:='=', ENO=>power, OUT=>P0_Start_Char:SMB88]  c3 ->
// row 4: c0 ^v  c2 [box]
// row 5: c0 ^v  c1 -(R) P0_Ctrl_Rcv_7:SM87.7, 1
// row 6: c0 ^v  c1 --  c2 [RCV EN:=power@row6, TBL:=VB100, PORT:=0, ENO=>power]  c3 ->
// row 7: c0 ^v  c2 [box]
// row 8: c0 ^  c1 --  c2 [XMT EN:=power@row8, TBL:=VB10, PORT:=0, ENO=>power]  c3 ->
// row 9: c2 [box]
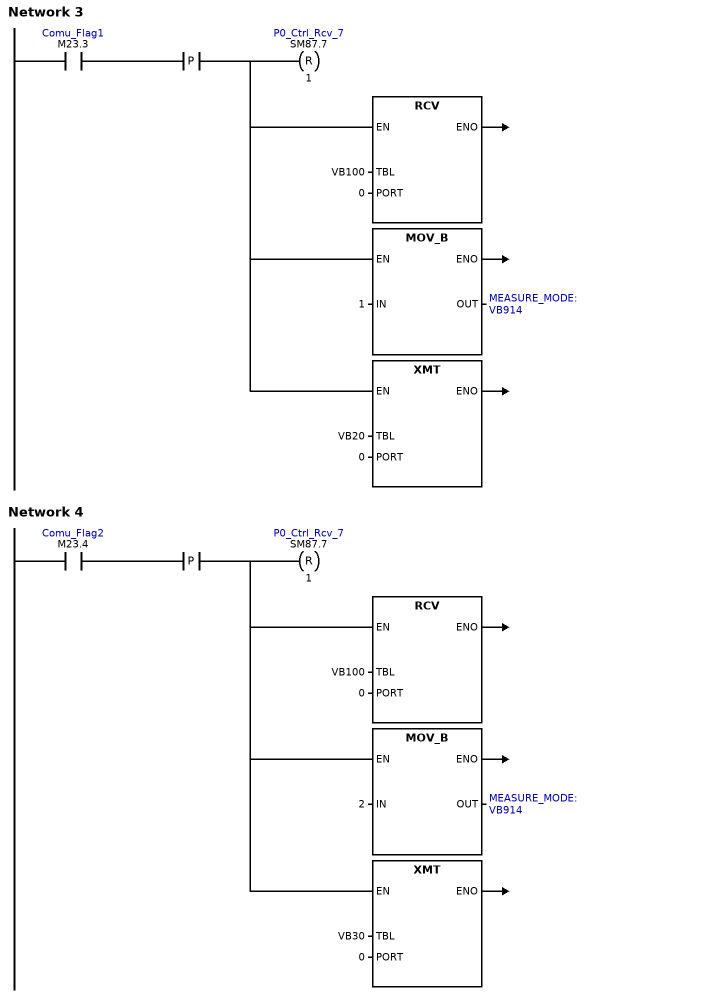
Network 3
// (network saved uncompiled; LAD cells follow)
// row 0: c0 -| |- Comu_Flag1:M23.3  c1 -|P|-  v  c2 -(R) P0_Ctrl_Rcv_7:SM87.7, 1
// row 1: c1 ^v  c2 --  c3 [RCV EN:=power@row1, TBL:=VB100, PORT:=0, ENO=>power]  c4 ->
// row 2: c1 ^v  c3 [box]
// row 3: c1 ^v  c2 --  c3 [MOV_B EN:=power@row3, IN:=1, ENO=>power, OUT=>MEASURE_MODE:VB914]  c4 ->
// row 4: c1 ^v  c3 [box]
// row 5: c1 ^  c2 --  c3 [XMT EN:=power@row5, TBL:=VB20, PORT:=0, ENO=>power]  c4 ->
// row 6: c3 [box]
Network 4
// (network saved uncompiled; LAD cells follow)
// row 0: c0 -| |- Comu_Flag2:M23.4  c1 -|P|-  v  c2 -(R) P0_Ctrl_Rcv_7:SM87.7, 1
// row 1: c1 ^v  c2 --  c3 [RCV EN:=power@row1, TBL:=VB100, PORT:=0, ENO=>power]  c4 ->
// row 2: c1 ^v  c3 [box]
// row 3: c1 ^v  c2 --  c3 [MOV_B EN:=power@row3, IN:=2, ENO=>power, OUT=>MEASURE_MODE:VB914]  c4 ->
// row 4: c1 ^v  c3 [box]
// row 5: c1 ^  c2 --  c3 [XMT EN:=power@row5, TBL:=VB30, PORT:=0, ENO=>power]  c4 ->
// row 6: c3 [box]
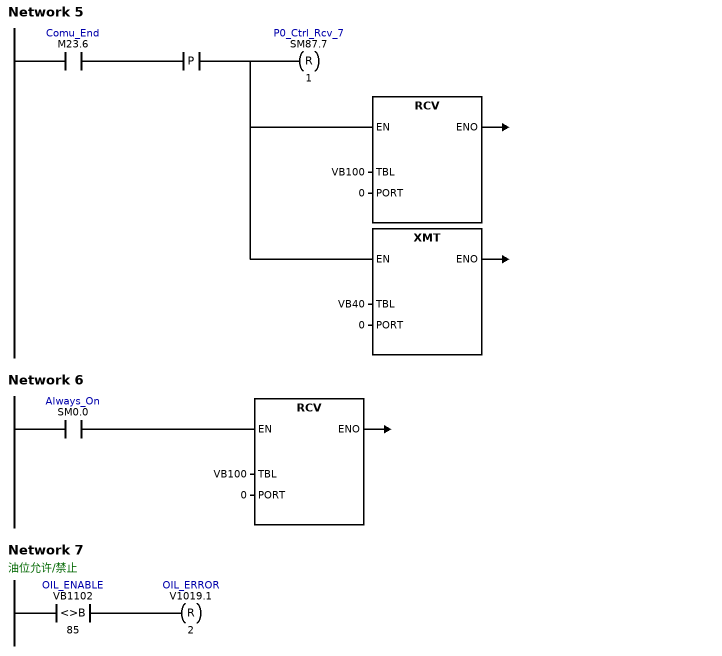
Network 5
// (network saved uncompiled; LAD cells follow)
// row 0: c0 -| |- Comu_End:M23.6  c1 -|P|-  v  c2 -(R) P0_Ctrl_Rcv_7:SM87.7, 1
// row 1: c1 ^v  c2 --  c3 [RCV EN:=power@row1, TBL:=VB100, PORT:=0, ENO=>power]  c4 ->
// row 2: c1 ^v  c3 [box]
// row 3: c1 ^  c2 --  c3 [XMT EN:=power@row3, TBL:=VB40, PORT:=0, ENO=>power]  c4 ->
// row 4: c3 [box]
Network 6
// (network saved uncompiled; LAD cells follow)
// row 0: c0 -| |- Always_On:SM0.0  c1 --  c2 [RCV EN:=power@row0, TBL:=VB100, PORT:=0, ENO=>power]  c3 ->
// row 1: c2 [box]
Network 7
// 油位允许/禁止
// (network saved uncompiled; LAD cells follow)
// row 0: c0 -|<>B|- OIL_ENABLE:VB1102, 85  c1 -(R) OIL_ERROR:V1019.1, 2
Network 8 // 网络标题
// 网络注释
END_SUBROUTINE_BLOCK

SUBROUTINE_BLOCK 初始化:SBR1
TITLE=
BEGIN
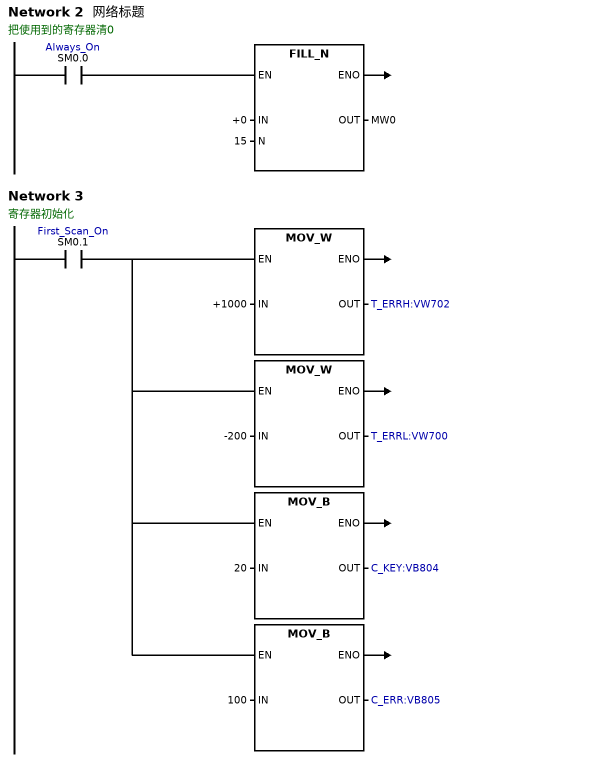
Network 2 // 网络标题
// 把使用到的寄存器清0
LD     Always_On:SM0.0
FILL   +0, MW0, 15
Network 3
// 寄存器初始化
LD     First_Scan_On:SM0.1
MOVW   +1000, T_ERRH:VW702
MOVW   -200, T_ERRL:VW700
MOVB   20, C_KEY:VB804
MOVB   100, C_ERR:VB805
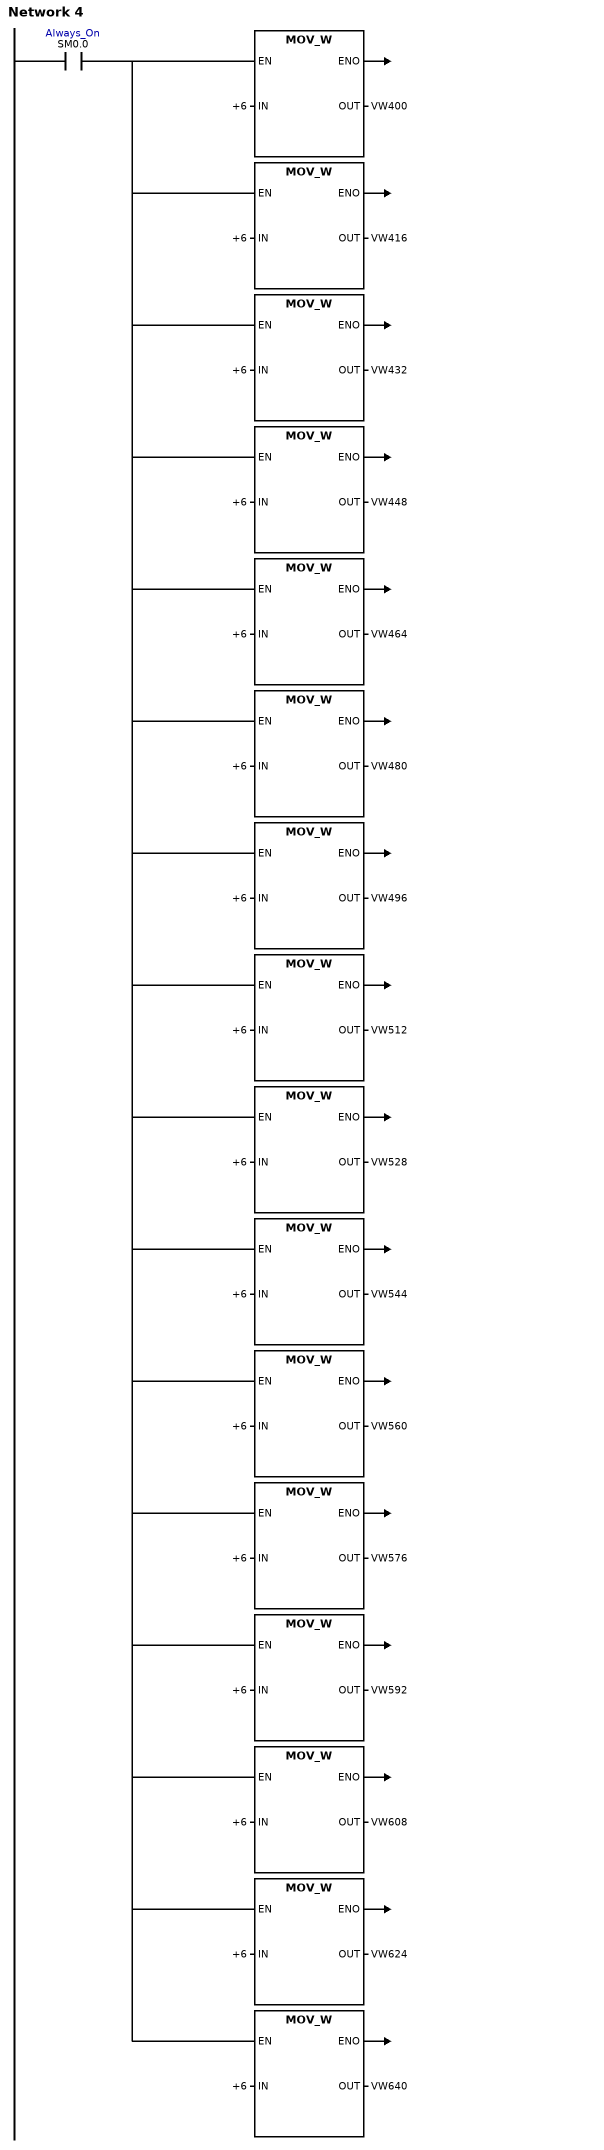
Network 4
LD     Always_On:SM0.0
MOVW   +6, VW400
MOVW   +6, VW416
MOVW   +6, VW432
MOVW   +6, VW448
MOVW   +6, VW464
MOVW   +6, VW480
MOVW   +6, VW496
MOVW   +6, VW512
MOVW   +6, VW528
MOVW   +6, VW544
MOVW   +6, VW560
MOVW   +6, VW576
MOVW   +6, VW592
MOVW   +6, VW608
MOVW   +6, VW624
MOVW   +6, VW640
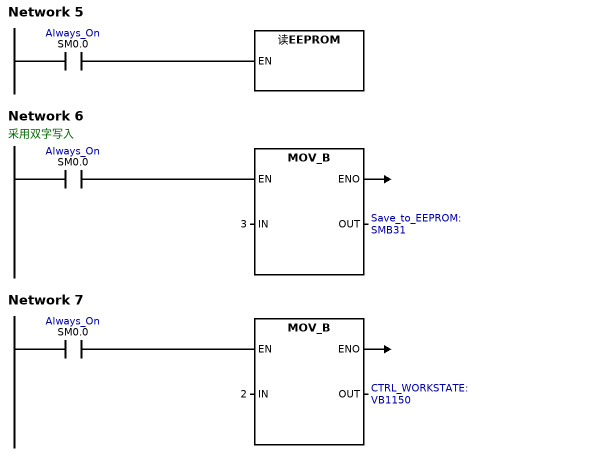
Network 5
LD     Always_On:SM0.0
CALL   读EEPROM:SBR8
Network 6
// 采用双字写入
LD     Always_On:SM0.0
MOVB   3, Save_to_EEPROM:SMB31
Network 7
LD     Always_On:SM0.0
MOVB   2, CTRL_WORKSTATE:VB1150
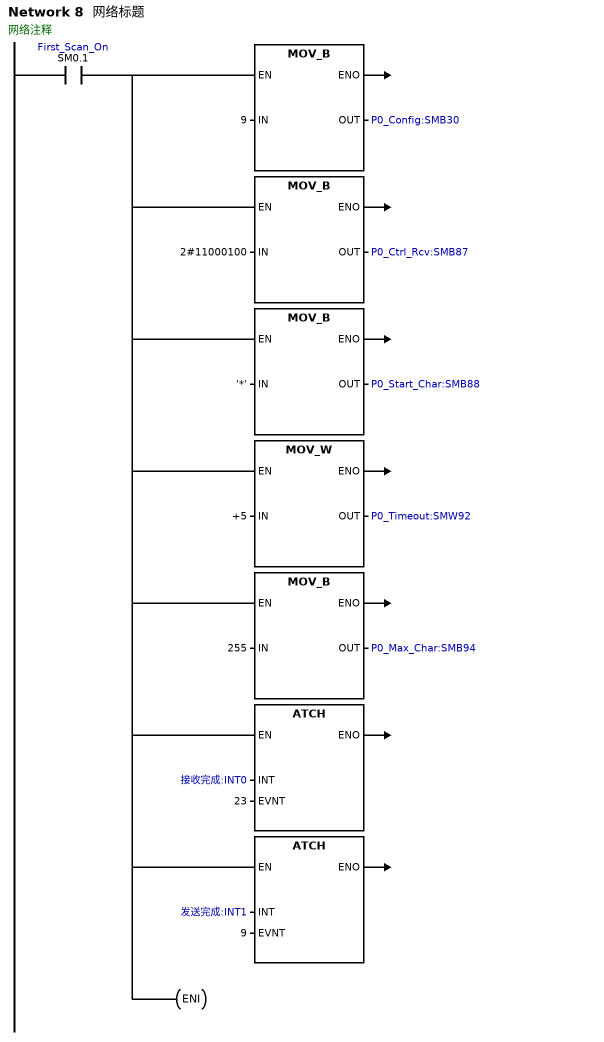
Network 8 // 网络标题
// 网络注释
LD     First_Scan_On:SM0.1
MOVB   9, P0_Config:SMB30
MOVB   2#11000100, P0_Ctrl_Rcv:SMB87
MOVB   '*', P0_Start_Char:SMB88
MOVW   +5, P0_Timeout:SMW92
MOVB   255, P0_Max_Char:SMB94
ATCH   接收完成:INT0, 23
ATCH   发送完成:INT1, 9
ENI
END_SUBROUTINE_BLOCK

SUBROUTINE_BLOCK 模块自动检测:SBR2
TITLE=
BEGIN
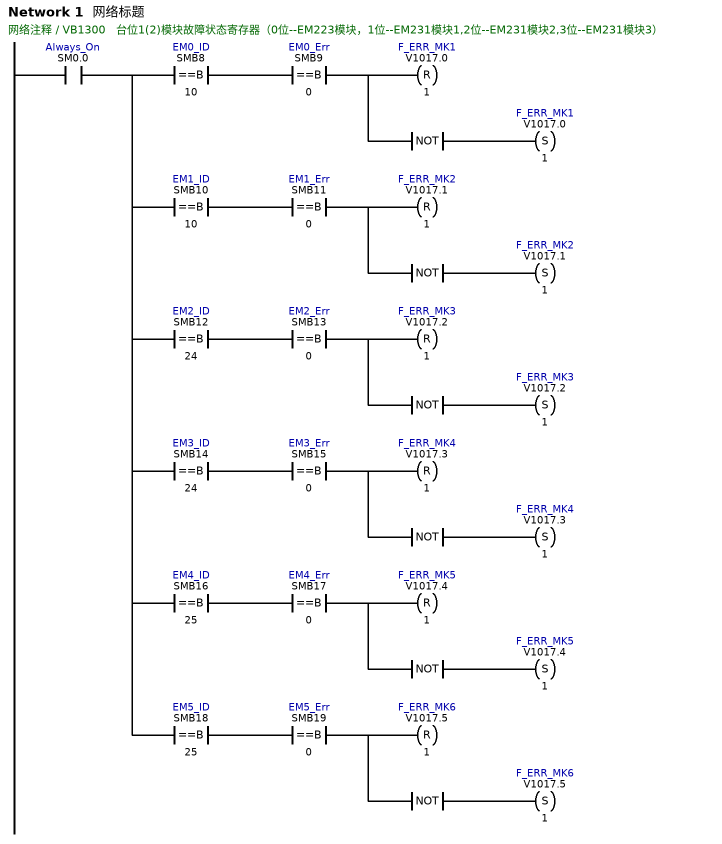
Network 1 // 网络标题
// 网络注释
// VB1300   台位1(2)模块故障状态寄存器（0位--EM223模块，1位--EM231模块1,2位--EM231模块2,3位--EM231模块3）
LD     Always_On:SM0.0
LPS
AB=    EM0_ID:SMB8, 10
AB=    EM0_Err:SMB9, 0
R      F_ERR_MK1:V1017.0, 1
NOT
S      F_ERR_MK1:V1017.0, 1
LRD
AB=    EM1_ID:SMB10, 10
AB=    EM1_Err:SMB11, 0
R      F_ERR_MK2:V1017.1, 1
NOT
S      F_ERR_MK2:V1017.1, 1
LRD
AB=    EM2_ID:SMB12, 24
AB=    EM2_Err:SMB13, 0
R      F_ERR_MK3:V1017.2, 1
NOT
S      F_ERR_MK3:V1017.2, 1
LRD
AB=    EM3_ID:SMB14, 24
AB=    EM3_Err:SMB15, 0
R      F_ERR_MK4:V1017.3, 1
NOT
S      F_ERR_MK4:V1017.3, 1
LRD
AB=    EM4_ID:SMB16, 25
AB=    EM4_Err:SMB17, 0
R      F_ERR_MK5:V1017.4, 1
NOT
S      F_ERR_MK5:V1017.4, 1
LPP
AB=    EM5_ID:SMB18, 25
AB=    EM5_Err:SMB19, 0
R      F_ERR_MK6:V1017.5, 1
NOT
S      F_ERR_MK6:V1017.5, 1
END_SUBROUTINE_BLOCK

SUBROUTINE_BLOCK 输入处理:SBR3
TITLE=
BEGIN
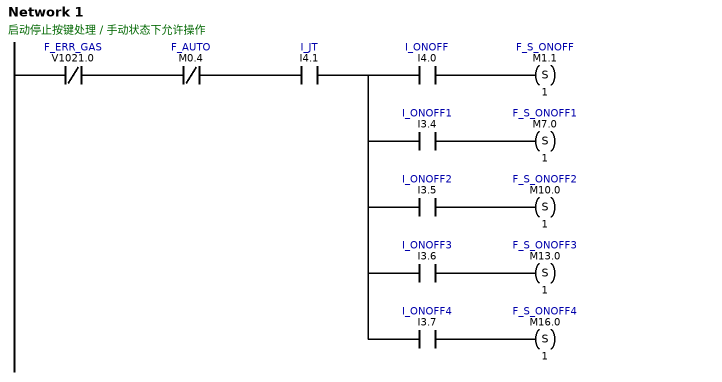
Network 1
// 启动停止按键处理
// 手动状态下允许操作
LDN    F_ERR_GAS:V1021.0
AN     F_AUTO:M0.4
A      I_JT:I4.1
LPS
A      I_ONOFF:I4.0
S      F_S_ONOFF:M1.1, 1
LRD
A      I_ONOFF1:I3.4
S      F_S_ONOFF1:M7.0, 1
LRD
A      I_ONOFF2:I3.5
S      F_S_ONOFF2:M10.0, 1
LRD
A      I_ONOFF3:I3.6
S      F_S_ONOFF3:M13.0, 1
LPP
A      I_ONOFF4:I3.7
S      F_S_ONOFF4:M16.0, 1
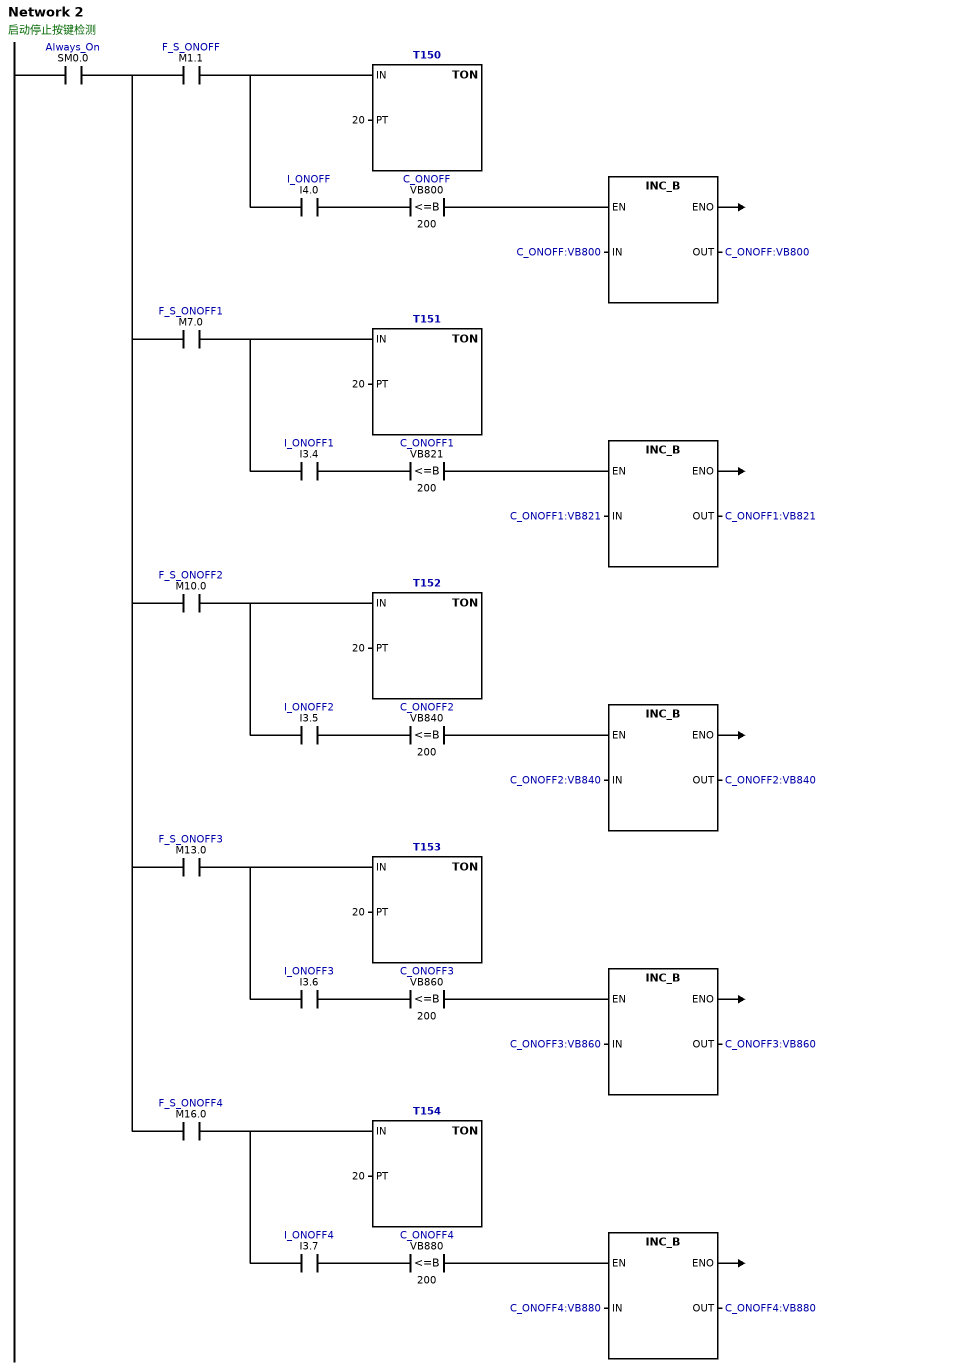
Network 2
// 启动停止按键检测
LD     Always_On:SM0.0
LPS
A      F_S_ONOFF:M1.1
TON    T150, 20
A      I_ONOFF:I4.0
AB<=   C_ONOFF:VB800, 200
INCB   C_ONOFF:VB800
LRD
A      F_S_ONOFF1:M7.0
TON    T151, 20
A      I_ONOFF1:I3.4
AB<=   C_ONOFF1:VB821, 200
INCB   C_ONOFF1:VB821
LRD
A      F_S_ONOFF2:M10.0
TON    T152, 20
A      I_ONOFF2:I3.5
AB<=   C_ONOFF2:VB840, 200
INCB   C_ONOFF2:VB840
LRD
A      F_S_ONOFF3:M13.0
TON    T153, 20
A      I_ONOFF3:I3.6
AB<=   C_ONOFF3:VB860, 200
INCB   C_ONOFF3:VB860
LPP
A      F_S_ONOFF4:M16.0
TON    T154, 20
A      I_ONOFF4:I3.7
AB<=   C_ONOFF4:VB880, 200
INCB   C_ONOFF4:VB880
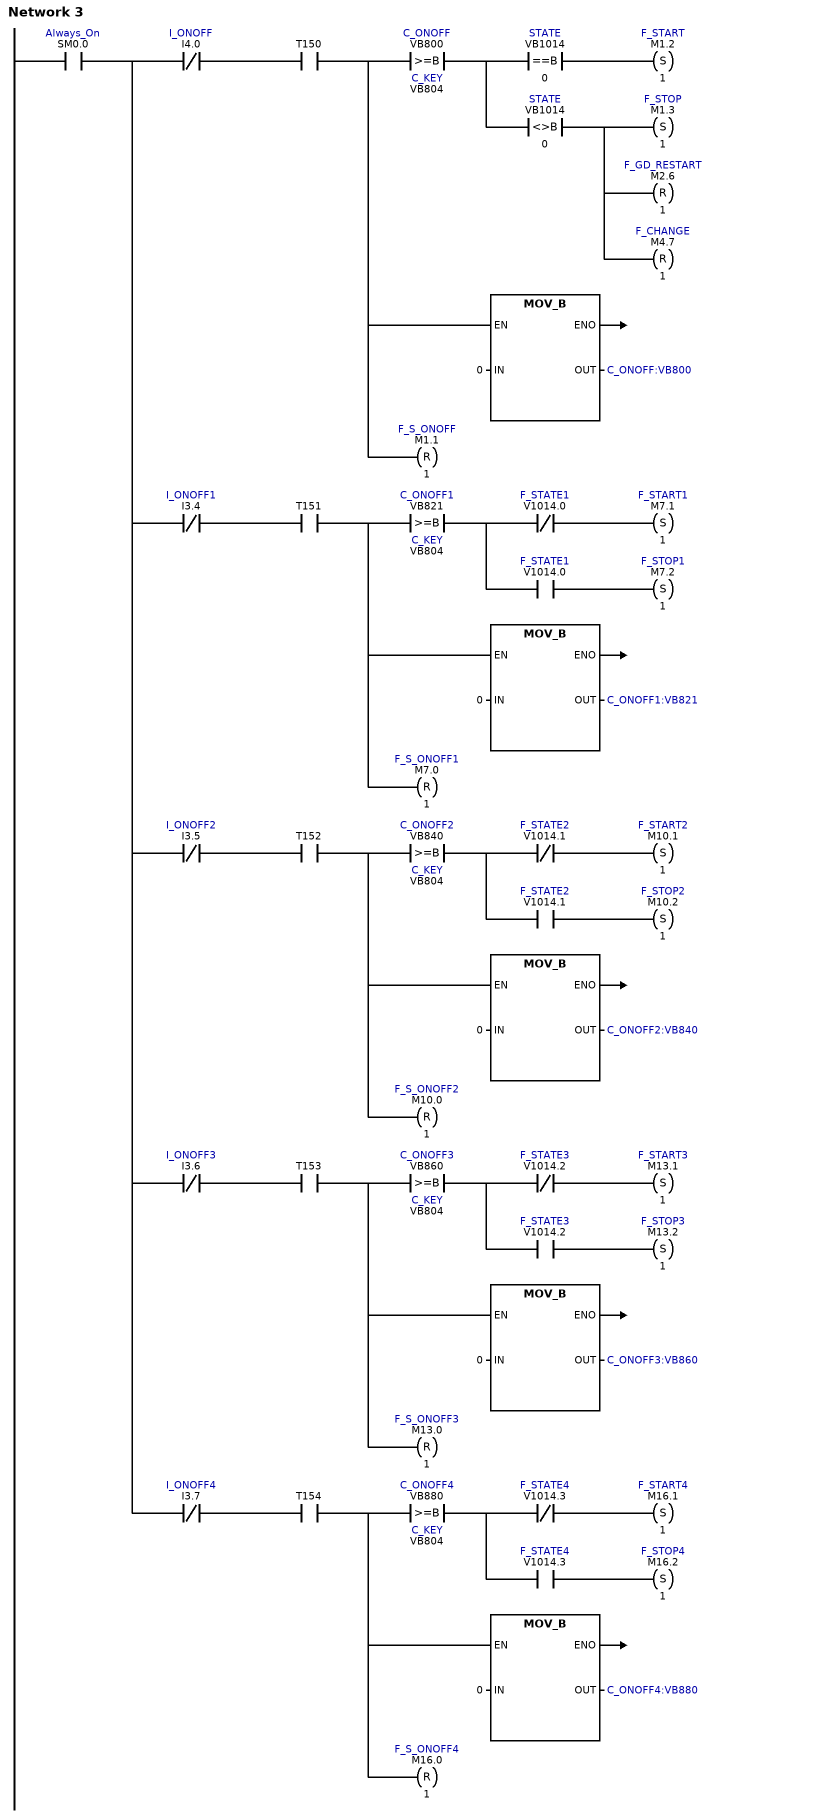
Network 3
LD     Always_On:SM0.0
LPS
AN     I_ONOFF:I4.0
A      T150
LPS
AB>=   C_ONOFF:VB800, C_KEY:VB804
LPS
AB=    STATE:VB1014, 0
S      F_START:M1.2, 1
LPP
AB<>   STATE:VB1014, 0
S      F_STOP:M1.3, 1
R      F_GD_RESTART:M2.6, 1
R      F_CHANGE:M4.7, 1
LPP
MOVB   0, C_ONOFF:VB800
R      F_S_ONOFF:M1.1, 1
LPP
LPS
AN     I_ONOFF1:I3.4
A      T151
LPS
AB>=   C_ONOFF1:VB821, C_KEY:VB804
LPS
AN     F_STATE1:V1014.0
S      F_START1:M7.1, 1
LPP
A      F_STATE1:V1014.0
S      F_STOP1:M7.2, 1
LPP
MOVB   0, C_ONOFF1:VB821
R      F_S_ONOFF1:M7.0, 1
LRD
AN     I_ONOFF2:I3.5
A      T152
LPS
AB>=   C_ONOFF2:VB840, C_KEY:VB804
LPS
AN     F_STATE2:V1014.1
S      F_START2:M10.1, 1
LPP
A      F_STATE2:V1014.1
S      F_STOP2:M10.2, 1
LPP
MOVB   0, C_ONOFF2:VB840
R      F_S_ONOFF2:M10.0, 1
LRD
AN     I_ONOFF3:I3.6
A      T153
LPS
AB>=   C_ONOFF3:VB860, C_KEY:VB804
LPS
AN     F_STATE3:V1014.2
S      F_START3:M13.1, 1
LPP
A      F_STATE3:V1014.2
S      F_STOP3:M13.2, 1
LPP
MOVB   0, C_ONOFF3:VB860
R      F_S_ONOFF3:M13.0, 1
LPP
AN     I_ONOFF4:I3.7
A      T154
LPS
AB>=   C_ONOFF4:VB880, C_KEY:VB804
LPS
AN     F_STATE4:V1014.3
S      F_START4:M16.1, 1
LPP
A      F_STATE4:V1014.3
S      F_STOP4:M16.2, 1
LPP
MOVB   0, C_ONOFF4:VB880
R      F_S_ONOFF4:M16.0, 1
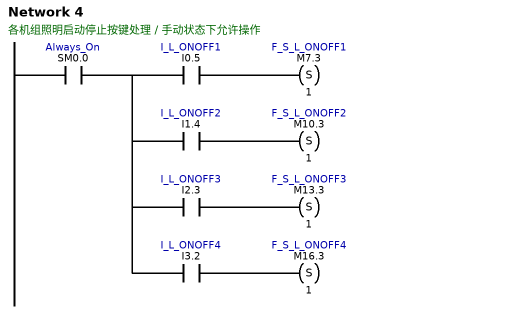
Network 4
// 各机组照明启动停止按键处理
// 手动状态下允许操作
LD     Always_On:SM0.0
LPS
A      I_L_ONOFF1:I0.5
S      F_S_L_ONOFF1:M7.3, 1
LRD
A      I_L_ONOFF2:I1.4
S      F_S_L_ONOFF2:M10.3, 1
LRD
A      I_L_ONOFF3:I2.3
S      F_S_L_ONOFF3:M13.3, 1
LPP
A      I_L_ONOFF4:I3.2
S      F_S_L_ONOFF4:M16.3, 1
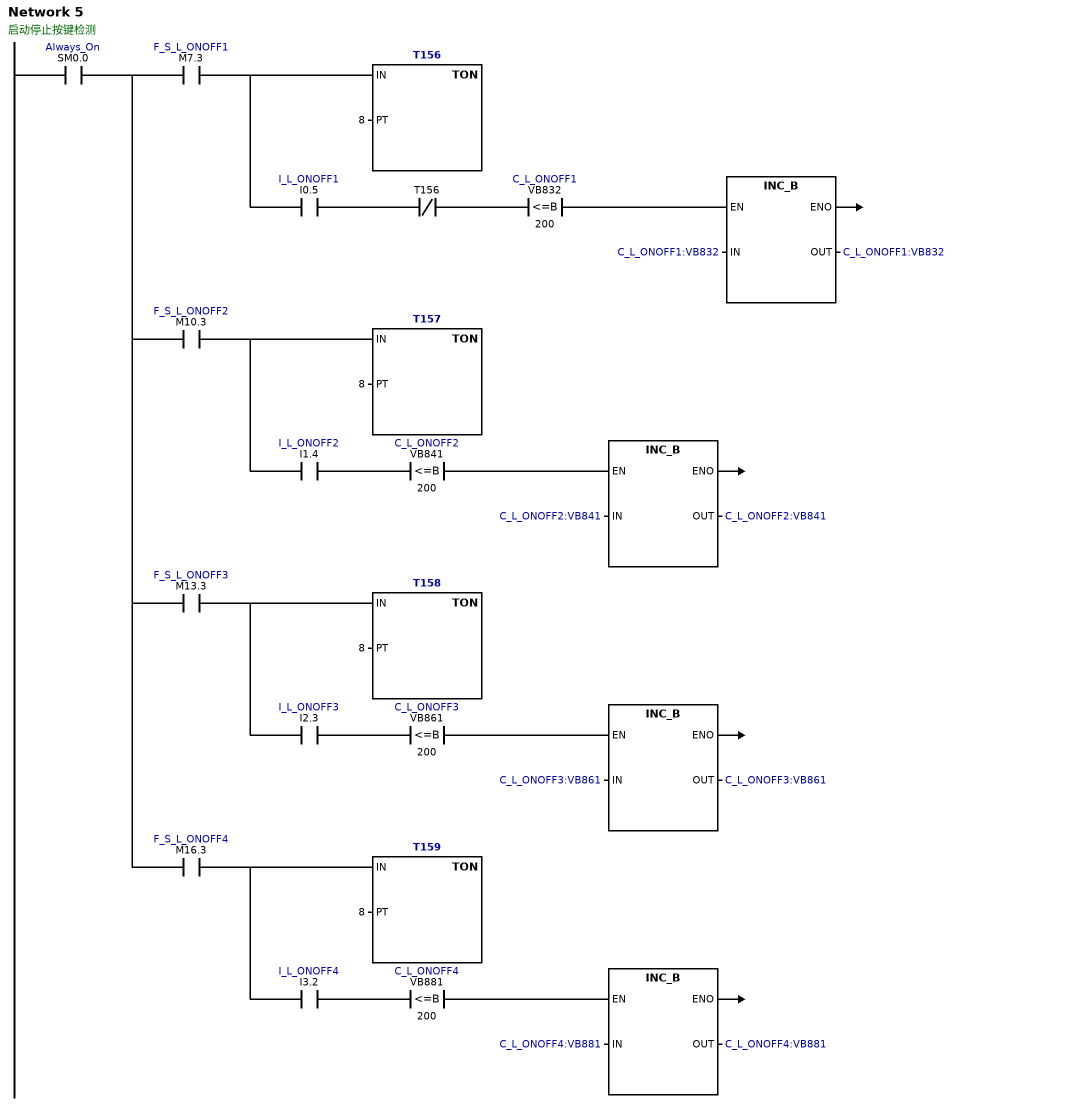
Network 5
// 启动停止按键检测
LD     Always_On:SM0.0
LPS
A      F_S_L_ONOFF1:M7.3
TON    T156, 8
A      I_L_ONOFF1:I0.5
AN     T156
AB<=   C_L_ONOFF1:VB832, 200
INCB   C_L_ONOFF1:VB832
LRD
A      F_S_L_ONOFF2:M10.3
TON    T157, 8
A      I_L_ONOFF2:I1.4
AB<=   C_L_ONOFF2:VB841, 200
INCB   C_L_ONOFF2:VB841
LRD
A      F_S_L_ONOFF3:M13.3
TON    T158, 8
A      I_L_ONOFF3:I2.3
AB<=   C_L_ONOFF3:VB861, 200
INCB   C_L_ONOFF3:VB861
LPP
A      F_S_L_ONOFF4:M16.3
TON    T159, 8
A      I_L_ONOFF4:I3.2
AB<=   C_L_ONOFF4:VB881, 200
INCB   C_L_ONOFF4:VB881
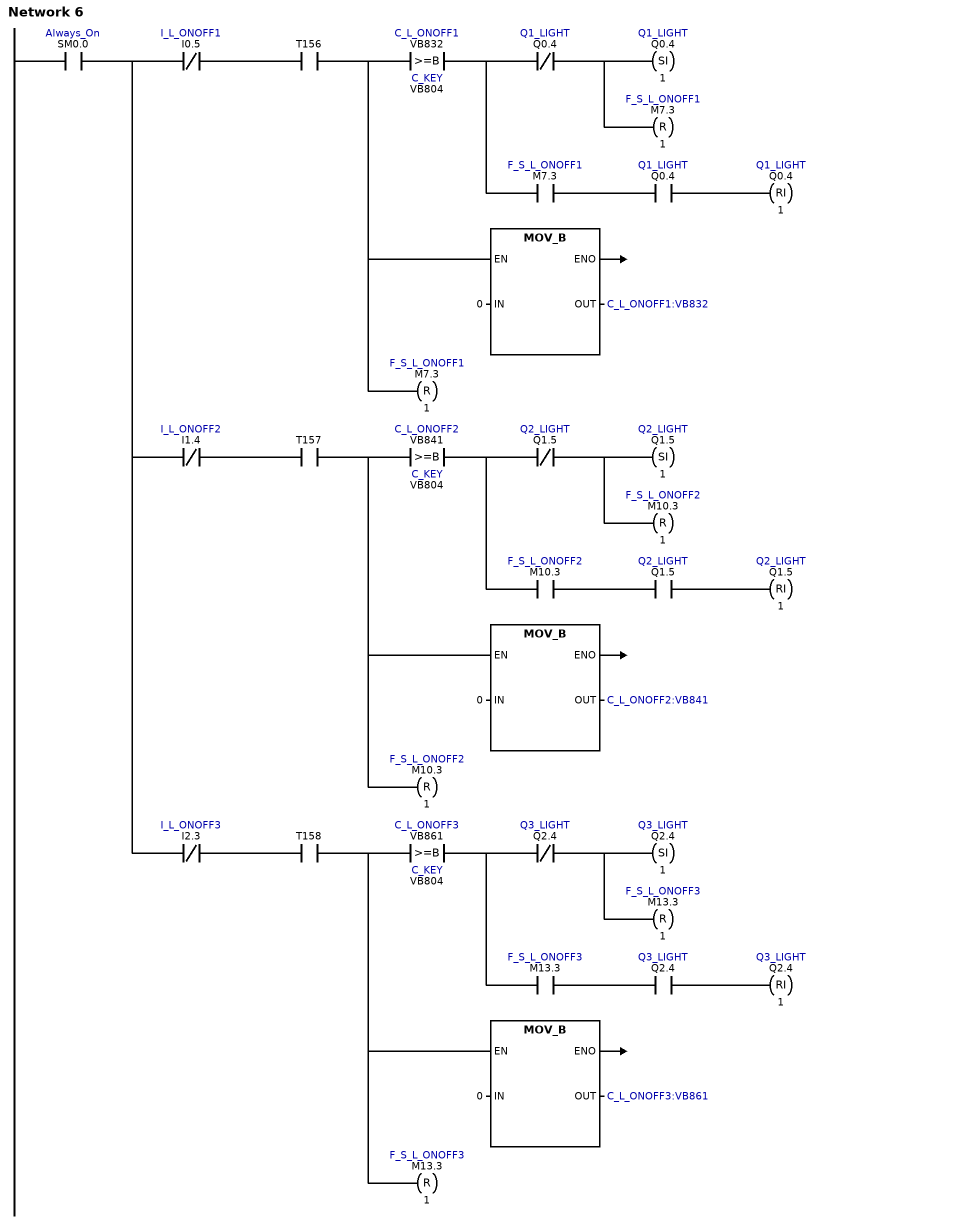
Network 6
LD     Always_On:SM0.0
LPS
AN     I_L_ONOFF1:I0.5
A      T156
LPS
AB>=   C_L_ONOFF1:VB832, C_KEY:VB804
LPS
AN     Q1_LIGHT:Q0.4
SI     Q1_LIGHT:Q0.4, 1
R      F_S_L_ONOFF1:M7.3, 1
LPP
A      F_S_L_ONOFF1:M7.3
A      Q1_LIGHT:Q0.4
RI     Q1_LIGHT:Q0.4, 1
LPP
MOVB   0, C_L_ONOFF1:VB832
R      F_S_L_ONOFF1:M7.3, 1
LRD
AN     I_L_ONOFF2:I1.4
A      T157
LPS
AB>=   C_L_ONOFF2:VB841, C_KEY:VB804
LPS
AN     Q2_LIGHT:Q1.5
SI     Q2_LIGHT:Q1.5, 1
R      F_S_L_ONOFF2:M10.3, 1
LPP
A      F_S_L_ONOFF2:M10.3
A      Q2_LIGHT:Q1.5
RI     Q2_LIGHT:Q1.5, 1
LPP
MOVB   0, C_L_ONOFF2:VB841
R      F_S_L_ONOFF2:M10.3, 1
LPP
AN     I_L_ONOFF3:I2.3
A      T158
LPS
AB>=   C_L_ONOFF3:VB861, C_KEY:VB804
LPS
AN     Q3_LIGHT:Q2.4
SI     Q3_LIGHT:Q2.4, 1
R      F_S_L_ONOFF3:M13.3, 1
LPP
A      F_S_L_ONOFF3:M13.3
A      Q3_LIGHT:Q2.4
RI     Q3_LIGHT:Q2.4, 1
LPP
MOVB   0, C_L_ONOFF3:VB861
R      F_S_L_ONOFF3:M13.3, 1
